    PERS robtarget YM61S:=[[-152,-102.434,331.364],[0.59149,-0.387784,-0.59121,0.3876],[-1,1,-3,0],[9E+09,8.10884,-48.3912,9E+09,9E+09,9E+09]];
    PERS robtarget YM61E:=[[-152,-136.732,324.386],[0.59149,-0.387784,-0.59121,0.3876],[-1,1,-3,0],[9E+09,8.10884,-48.3912,9E+09,9E+09,9E+09]];
    PERS robtarget YM62S:=[[-152,-143.638,394.581],[0.591293,-0.387692,-0.591403,0.387699],[-1,1,-3,0],[9E+09,7.68338,-48.3166,9E+09,9E+09,9E+09]];
    PERS robtarget YM62E:=[[-152,-165.995,387.902],[0.591293,-0.387692,-0.591403,0.387699],[-1,1,-3,0],[9E+09,7.68338,-48.3166,9E+09,9E+09,9E+09]];
    PERS robtarget YM63S:=[[-152,-136.961,363.19],[0.65293,-0.271555,-0.652826,0.271586],[-1,1,-3,0],[9E+09,9.82577,-48.6742,9E+09,9E+09,9E+09]];
    PERS robtarget YM63E:=[[-152,-158.994,355.019],[0.65293,-0.271555,-0.652826,0.271586],[-1,1,-3,0],[9E+09,9.82577,-48.6742,9E+09,9E+09,9E+09]];
    PERS robtarget YM67S:=[[-152,-100.439,322.029],[0.65293,-0.271555,-0.652826,0.271586],[-1,1,-3,0],[9E+09,8.96447,-48.5355,9E+09,9E+09,9E+09]];
    PERS robtarget YM67E:=[[-152,-134.61,314.453],[0.65293,-0.271555,-0.652826,0.271586],[-1,1,-3,0],[9E+09,8.96447,-48.5355,9E+09,9E+09,9E+09]];
    PERS robtarget YM66S:=[[-152,-225,411.8],[0.663642,-0.282382,-0.641613,0.261097],[-1,1,-3,0],[9E+09,7.65,-44.82,9E+09,9E+09,9E+09]];
    PERS robtarget YM66E:=[[-152,-189,411.8],[0.663642,-0.282382,-0.641613,0.261097],[-1,1,-3,0],[9E+09,7.65,-44.82,9E+09,9E+09,9E+09]];
    PERS robtarget YM65S:=[[-152,-225,411.8],[0.663642,-0.282382,-0.641613,0.261097],[-1,1,-3,0],[9E+09,7.65,-44.82,9E+09,9E+09,9E+09]];
    PERS robtarget YM65E:=[[-152,-189,411.8],[0.663642,-0.282382,-0.641613,0.261097],[-1,1,-3,0],[9E+09,7.65,-44.82,9E+09,9E+09,9E+09]];
    PERS robtarget YM64S:=[[-152,-225,411.8],[0.663642,-0.282382,-0.641613,0.261097],[-1,1,-3,0],[9E+09,7.65,-44.82,9E+09,9E+09,9E+09]];
    PERS robtarget YM64E:=[[-152,-189,411.8],[0.663642,-0.282382,-0.641613,0.261097],[-1,1,-3,0],[9E+09,7.65,-44.82,9E+09,9E+09,9E+09]];
    PERS robtarget YM64KS:=[[-152,-236.712,697.465],[0.65293,-0.271555,-0.652826,0.271586],[-1,1,-3,0],[9E+09,1.26795,-46.7321,9E+09,9E+09,9E+09]];
    PERS robtarget YM64KE:=[[-152,-260.629,694.325],[0.65293,-0.271555,-0.652826,0.271586],[-1,1,-3,0],[9E+09,1.26795,-46.7321,9E+09,9E+09,9E+09]];
    PERS robtarget YM65KS:=[[-152,-226.703,599.049],[0.65293,-0.271555,-0.652826,0.271586],[-1,1,-3,0],[9E+09,6,-48,9E+09,9E+09,9E+09]];
    PERS robtarget YM65KE:=[[-152,-249.965,589.663],[0.65293,-0.271555,-0.652826,0.271586],[-1,1,-3,0],[9E+09,6,-48,9E+09,9E+09,9E+09]];
    PERS robtarget YM66KS:=[[-152,-204.477,493.494],[0.65293,-0.271555,-0.652826,0.271586],[-1,1,-3,0],[9E+09,11.127,-48.873,9E+09,9E+09,9E+09]];
    PERS robtarget YM66KE:=[[-152,-226.433,477.965],[0.65293,-0.271555,-0.652826,0.271586],[-1,1,-3,0],[9E+09,11.127,-48.873,9E+09,9E+09,9E+09]];
    PERS robtarget YM67KS:=[[-152,-206.596,501.506],[0.65293,-0.271555,-0.652826,0.271586],[-1,1,-3,0],[9E+09,10.6921,-48.8079,9E+09,9E+09,9E+09]];
    PERS robtarget YM67KE:=[[-152,-228.685,486.483],[0.65293,-0.271555,-0.652826,0.271586],[-1,1,-3,0],[9E+09,10.6921,-48.8079,9E+09,9E+09,9E+09]];
    PERS robtarget YM68S:=[[-152,-131.055,340.199],[0.653753,-0.269329,-0.653858,0.269329],[-1,1,-3,0],[9E+09,11.563,-48.937,9E+09,9E+09,9E+09]];
    PERS robtarget YM68E:=[[-152,-152.782,330.846],[0.653753,-0.269329,-0.653858,0.269329],[-1,1,-3,0],[9E+09,11.563,-48.937,9E+09,9E+09,9E+09]];
    PERS robtarget YM69S:=[[-152,-97.8611,310.69],[0.65091,-0.275923,-0.651211,0.275876],[-1,1,-3,0],[9E+09,9.82577,-48.6742,9E+09,9E+09,9E+09]];
    PERS robtarget YM69E:=[[-152,-131.894,302.519],[0.65091,-0.275923,-0.651211,0.275876],[-1,1,-3,0],[9E+09,9.82577,-48.6742,9E+09,9E+09,9E+09]];

    PERS robtarget XM69S:=[[-51.74,-38.43,346.47],[0.69982,-0.714319,-0.000177661,-0.000168257],[0,-1,-1,0],[9E+09,9.82577,-48.6742,9E+09,9E+09,9E+09]];
    PERS robtarget XM69E:=[[-81.74,-44.99,332.86],[0.69982,-0.714319,-0.000177665,-0.000168594],[0,-1,-1,0],[9E+09,9.82577,-48.6742,9E+09,9E+09,9E+09]];
    PERS pose SRM69X:=[[-0.305832,0.0427742,0.000274658],[1,0,0,0]];

    PERS robtarget XM61S:=[[-51.74,-14.78,-164.74],[0.707159,-0.707055,-0.000176256,-0.000169845],[-1,1,-2,0],[9E+09,8.10884,-48.3912,9E+09,9E+09,9E+09]];
    PERS robtarget XM61E:=[[-81.74,-4.2,65],[0.707159,-0.707055,-0.000175884,-0.000170178],[-1,0,-1,0],[9E+09,8.10884,-48.3912,9E+09,9E+09,9E+09]];
    PERS pose SRM61X:=[[1.22222,0.048152,0.00824738],[1,0,0,0]];

    PERS robtarget YM69air0:=[[323.43,-909.32,657.88],[0.75163,-0.489467,-0.418492,0.142614],[-1,1,-3,0],[9E+09,0,-45,9E+09,9E+09,9E+09]];
    PERS robtarget YM69air1:=[[741.26,-226.51,717.48],[0.702088,-0.433242,-0.448105,0.344349],[-1,1,-3,0],[9E+09,0,-45,9E+09,9E+09,9E+09]];
    PERS robtarget YM69air2:=[[-25.10,218.09,408.29],[0.758077,-0.477323,-0.345026,0.280071],[0,2,-3,0],[9E+09,-7.75,-44.65,9E+09,9E+09,9E+09]];

    PERS robtarget XM49S:=[[-51,-69.7,-355.45],[0.00026471,0.974449,-0.224609,-3.1544E-05],[-1,0,0,0],[9E+09,-18.2042,-49.7958,9E+09,9E+09,9E+09]];
    PERS robtarget XM49E:=[[-81.8,-49.99,-284],[0.674318,-0.67636,0.209812,0.209312],[0,-1,0,0],[9E+09,-18.2042,-49.7958,9E+09,9E+09,9E+09]];
    PERS pose SRM49X:=[[1.06467,0.0033226,3.05176E-05],[1,0,0,0]];

    PERS robtarget YM41air0:=[[322.86,-786.84,1283.97],[0.75163,-0.489467,-0.418492,0.142614],[-1,1,-3,0],[9E+09,0,0,9E+09,9E+09,9E+09]];
    PERS robtarget YM41air1:=[[438.12,-1.09,1129.17],[0.714752,-0.443018,-0.427615,0.331677],[-1,1,-3,0],[9E+09,-7.75,-44.64,9E+09,9E+09,9E+09]];
    PERS robtarget YM41air2:=[[280.06,246.13,1162.64],[0.711624,-0.440596,-0.432799,0.334891],[-1,1,-3,0],[9E+09,-7.75,-44.65,9E+09,9E+09,9E+09]];


    PERS robtarget XM69air1:=[[406.95,-323.45,691.79],[0.681158,-0.726208,-0.091705,-0.0152943],[-1,1,-2,0],[9E+09,0,0,9E+09,9E+09,9E+09]];
    PERS robtarget XM69air2:=[[201.71,-906.55,542.23],[0.865261,-0.501321,-0.00012615,-0.00020979],[-1,-1,-1,0],[9E+09,0,-45,9E+09,9E+09,9E+09]];
    PERS robtarget XM69air3:=[[201.99,-627.42,55.34],[0.865261,-0.501321,-0.000126247,-0.000209686],[0,-1,-1,0],[9E+09,18.6523,-49.8477,9E+09,9E+09,9E+09]];
CONST robtarget XM69air13:=[[466.38,-593.12,1090.02],[0.546463,0.569613,0.0273419,-0.61333],[-1,2,-5,0],[9E+09,-7.78641E-06,6.55343E-08,9E+09,9E+09,9E+09]];
CONST robtarget XM41air13:=[[343.43,-602.92,741.89],[0.834426,0.42267,-0.338231,-0.103362],[-1,1,-4,0],[9E+09,-0.487862,-2.87448,9E+09,9E+09,9E+09]];
CONST robtarget XM41air14:=[[379.39,-439.44,917.00],[0.800618,0.381354,-0.240244,-0.394798],[-1,-2,0,0],[9E+09,-0.335924,-1.97573,9E+09,9E+09,9E+09]];
PERS robtarget pathomestnatneg45degrees:=[[1642.08,-1115.70,2682.87],[0.0875938,-0.425292,0.894504,0.106378],[-1,0,-2,0],[9E+09,-3.62032,-44.8189,9E+09,9E+09,9E+09]];
PERS robtarget A30air20:=[[382.75,-479.80,640.65],[0.391305,-0.39464,-0.584209,0.591473],[-1,0,-1,0],[9E+09,5.5,-135,9E+09,9E+09,9E+09]];
PERS robtarget B33air30:=[[-67.79,-632.04,318.04],[0.164585,0.515201,-0.472181,0.696079],[-1,1,-3,0],[9E+09,-13.5,136.5,9E+09,9E+09,9E+09]];
PERS robtarget B33air40:=[[-323.48,-348.44,373.29],[0.122788,0.72187,-0.311157,0.605812],[-1,1,-3,0],[9E+09,0,135,9E+09,9E+09,9E+09]];
PERS robtarget AIRTOANCH3:=[[-8.6,-155.14,117.47],[0.263609,-0.696089,0.660491,-0.0985977],[-1,1,-2,0],[9E+09,-40,100,9E+09,9E+09,9E+09]];
PERS robtarget H18AIRTOYL69S4:=[[204.19,-4.45,429.35],[0.341759,0.582985,-0.611047,-0.412252],[-1,1,-1,0],[9E+09,13.0111,44.6842,9E+09,9E+09,9E+09]];
PERS robtarget H18AIRTOG40_1:=[[426.16,1.81,851.86],[0.361748,-0.776477,-0.217756,0.467765],[-1,2,-2,0],[9E+09,-20,-50,9E+09,9E+09,9E+09]];

PERS robtarget XL4air23:=[[691.52,-162.97,1726.77],[0.491618,-0.102439,-0.167584,-0.848371],[-1,2,0,0],[9E+09,-10.15,44.19,9E+09,9E+09,9E+09]];
CONST robtarget AIRTOT30_10:=[[762.15,413.99,710.03],[0.077116,-0.841504,-0.161316,0.509805],[0,2,-3,0],[9E+09,-24.4581,-62.5826,9E+09,9E+09,9E+09]];
PERS robtarget F90AIRTOG40_1:=[[723.59,171.68,1587.9],[0.0227694,0.706641,-0.0229355,-0.706834],[-1,2,-2,0],[9E+09,-26,-45,9E+09,9E+09,9E+09]];

    PERS robtarget XM4air23:=[[679.92,-287.42,2151.86],[0.491619,-0.10244,-0.167584,-0.848371],[-1,1,0,0],[9E+09,0,45,9E+09,9E+09,9E+09]];

    CONST robtarget YL69air3:=[[575.73,-240.27,159.13],[0.142157,0.421918,-0.892494,-0.0723355],[-1,1,-1,0],[9E+09,12.7709,44.9833,9E+09,9E+09,9E+09]];
    CONST robtarget M49air5:=[[67.09,-478.73,-557.98],[0.703183,-0.592785,-0.0745474,0.385464],[-1,-1,0,0],[9E+09,-22,-39,9E+09,9E+09,9E+09]];
    CONST robtarget B35air_1:=[[-118.21,-790.16,748.75],[0.222108,0.671312,-0.312762,0.634183],[-1,0,-3,0],[9E+09,-14.37,135,9E+09,9E+09,9E+09]];
    CONST robtarget B35air_2:=[[-474.04,-451.28,796.03],[0.222108,0.671312,-0.312762,0.634183],[-1,0,-2,0],[9E+09,-14.37,135,9E+09,9E+09,9E+09]];
    CONST robtarget A32air_1:=[[514.14,-702.66,989.84],[0.405528,-0.370817,-0.574896,0.606248],[-1,0,-1,0],[9E+09,-1.37,-125,9E+09,9E+09,9E+09]];
    CONST robtarget A32air_2:=[[289.83,-781.28,1194.82],[0.36389,-0.403742,-0.562005,0.62348],[-1,0,-1,0],[9E+09,-1.37,-125,9E+09,9E+09,9E+09]];
    CONST robtarget B32air_1:=[[-490.20,-367.22,1109.93],[0.274121,0.675425,-0.244148,0.639571],[-1,0,-2,0],[9E+09,-5.48905,135.061,9E+09,9E+09,9E+09]];
    CONST robtarget B32air_2:=[[-137.07,-805.28,1092.89],[0.265044,0.655577,-0.224708,0.67043],[-1,0,-3,0],[9E+09,0.207107,134.293,9E+09,9E+09,9E+09]];
    CONST robtarget pjhomeSTN1zeroand180degrees:=[[1508.32,-0.13,3794.95],[0.2896,-0.00402012,0.957097,-0.0089805],[0,-1,-1,0],[9E+09,-0.0499035,180.021,9E+09,9E+09,9E+09]];
    CONST robtarget VRL52:=[[22.52,-205.94,976.00],[0.523446,-0.751557,0.24068,-0.321309],[-1,1,-2,0],[9E+09,-14.1988,49.3012,9E+09,9E+09,9E+09]];
    CONST robtarget VRM58:=[[-91.58,-127.90,952.71],[0.596926,-0.358375,-0.702933,-0.145368],[-1,0,-2,0],[9E+09,-14.1988,-49.3012,9E+09,9E+09,9E+09]];
    CONST robtarget VRG37:=[[1759.44,-115.82,2299.26],[0.0849098,0.0286926,0.995945,0.00776692],[-1,1,-2,0],[9E+09,-4.82784,-44.5104,9E+09,9E+09,9E+09]];
    CONST robtarget pzerostn194:=[[97.93,1457.09,1662.03],[0.650331,-0.0562801,-0.749121,-0.112781],[0,0,0,0],[9E+09,-0.00693957,94.0524,9E+09,9E+09,9E+09]];
    PERS robtarget pairtoL46_1:=[[191.64,-867.11,2097.29],[0.475472,-0.804215,0.076122,0.348382],[-1,-1,0,0],[9E+09,-22,-39,9E+09,9E+09,9E+09]];
    PERS robtarget XA3010:=[[682.98,-298.39,1395.43],[0.907863,-0.162432,0.0630474,0.381348],[-1,-1,-1,0],[9E+09,-10,-120,9E+09,9E+09,9E+09]];
    CONST robtarget YL69air10:=[[-200.13,-1122.9,1105.9],[0.0565202,0.961932,-0.056947,0.261247],[-1,0,-2,0],[9E+09,-10.15,44.19,9E+09,9E+09,9E+09]];
    PERS robtarget AG103danger:=[[98.44,-98.06,-251.18],[0.197528,-0.384452,-0.0264323,-0.901377],[-1,1,-3,0],[9E+09,35,102,9E+09,9E+09,9E+09]];
    PERS num limit:=-42;
    PERS robtarget R100:=[[-101.31,-14.09,-203.92],[0.000217526,0.000217373,0.707106,-0.707108],[-1,1,-3,0],[9E+09,33.5,180,9E+09,9E+09,9E+09]];

    PERS num ADJTIPSRCH:=-0.00275073;
    PERS num WTIPANGLEadj:=21.5028;
    PERS pose SRaveofG11G12:=[[0,-0.0110421,0],[1,0,0,0]];


!!!!!!these are declarations for 18H family of tips!!!!!!
    PERS pose SRTIPY18HL:=[[0,0,0],[1,0,0,0]];
    PERS pose SRTIPY18HR:=[[0,0,0],[1,0,0,0]];
	CONST robtarget SPTIPY18HLE:=[[38.00,-12.70,230.00],[0.500261,-0.499982,-0.499745,0.500012],[0,1,-2,0],[9E+09,0,-90,9E+09,9E+09,9E+09]];
	CONST robtarget SPTIPY18HRE:=[[-38.00,-12.70,230.00],[0.500261,-0.499982,0.499745,-0.500012],[0,2,-3,0],[9E+09,0,90,9E+09,9E+09,9E+09]];

	CONST robtarget SPU600HLE:=[[38,-16.5,230],[0.500261,-0.499982,-0.499745,0.500012],[0,1,-2,0],[9E+09,0,-90,9E+09,9E+09,9E+09]];
	CONST robtarget SPU650HRE:=[[-38,-16.5,230],[0.500261,-0.499982,0.499745,-0.500012],[0,2,-3,0],[9E+09,0,90,9E+09,9E+09,9E+09]];

    PERS robtarget halfwayhome_M:=[[323.43,-909.32,657.88],[0.75163,-0.489467,-0.418492,0.142614],[-1,0,-2,0],[9E+09,0,-45,9E+09,9E+09,9E+09]];
    PERS robtarget halfwayhome_L:=[[285.94,-356.45,959.29],[0.0234875,-0.737204,0.674708,-0.0273506],[-1,0,-1,0],[9E+09,0,45,9E+09,9E+09,9E+09]];
    PERS robtarget halfwayhome_A:=[[496.89,-178.24,594.79],[0.00515288,-0.986648,-0.155581,-0.0479021],[-1,2,-2,1],[9E+09,0,-135,9E+09,9E+09,9E+09]];
    PERS robtarget halfwayhome_B:=[[-434.18,-117.02,196.36],[0.0151057,0.00487122,0.994314,0.105302],[0,1,-1,0],[9E+09,0,135,9E+09,9E+09,9E+09]];
    PERS robtarget halfwayhome_G:=[[-643.51,-162.5,668.83],[0.0892073,-0.589525,0.793761,-0.120189],[-1,0,0,0],[9E+09,0,45,9E+09,9E+09,9E+09]];
    PERS robtarget halfwayhome_H:=[[780.67,-310.30,634.14],[0.236488,0.969948,0.0278582,0.0499801],[-1,1,-1,0],[9E+09,0,-45,9E+09,9E+09,9E+09]];

    PERS robtarget Troot1:=[[99.82,-61.36,159.35],[0.627626,-0.443283,-0.355925,-0.531886],[-1,0,-2,0],[9E+09,42,0,9E+09,9E+09,9E+09]];
    PERS robtarget Troot2:=[[-93.69,-61.65,160.34],[0.627627,-0.443282,-0.355926,-0.531886],[-1,0,-2,0],[9E+09,42,-7.12501E-05,9E+09,9E+09,9E+09]];

    CONST num FBfirst:=-17;
    CONST num FBsecond:= -11;

!!!!!!!!!!!!!!!!!!!!!!!!!!!!!!!!!!!END OF DECLARATIONS      !!!!!!!!!!!!!!!!!!!!!!!!!!!!!!

    CONST robtarget pat45negair1:=[[380.92,-801.85,1168.30],[0.000430871,-0.974447,0.224617,-5.83607E-05],[-1,0,0,0],[9E+09,0,-45,9E+09,9E+09,9E+09]];

    CONST robtarget AIRU1:=[[144.96,-753.41,659.47],[0.235813,-0.732282,-0.251047,0.587478],[0,2,-3,0],[9E+09,-7.00985,-63.2077,9E+09,9E+09,9E+09]];
    PERS robtarget SPUY33E:=[[-170.365,-78.7078,203.558],[0.510017,0.49007,-0.509654,-0.489864],[0,0,-3,0],[9E+09,27.0001,-45.0004,9E+09,9E+09,9E+09]];
    PERS robtarget SPUX33E:=[[-124.148,-21.7897,284.454],[0.49981,-0.500212,-0.4998,-0.500178],[-1,0,-2,0],[9E+09,27.0001,-45,9E+09,9E+09,9E+09]];
    PERS robtarget SPTY33E:=[[150.444,-80.007,203.769],[0.494322,-0.505307,0.494754,-0.505499],[0,4,-5,0],[9E+09,27,45.0002,9E+09,9E+09,9E+09]];
    PERS robtarget SPTX33E:=[[120.8,-22.1731,284.337],[0.502915,-0.503196,-0.49696,-0.496892],[-1,1,-3,0],[9E+09,26.9999,45.0001,9E+09,9E+09,9E+09]];

    PERS robtarget SPUY36E:=[[-172.488,-16.8208,232.206],[0.632719,-0.315721,-0.632589,0.315941],[0,0,-1,0],[9E+09,-15.9999,-135,9E+09,9E+09,9E+09]];
    PERS robtarget SPUX36E:=[[-142.33,-74.3,308.23],[0.6415,-0.26243,-0.650252,-0.311097],[-1,0,-2,0],[9E+09,22,-48.8794,9E+09,9E+09,9E+09]];
    PERS robtarget SPTY36E:=[[171.992,-18.0388,231.844],[0.315314,0.632751,0.315517,0.632971],[0,1,-3,0],[9E+09,-15.9999,-225,9E+09,9E+09,9E+09]];
    PERS robtarget SPTX36E:=[[142.09,-74.99,306.8],[0.313457,-0.650452,-0.267257,-0.638146],[-1,1,-2,0],[9E+09,22,48.0666,9E+09,9E+09,9E+09]];

    PERS robtarget SPUZ33E:=[[-86.4363,-72.1286,298.144],[0.606826,-0.362533,-0.518582,-0.481046],[-1,0,-2,0],[9E+09,27,-45.0002,9E+09,9E+09,9E+09]];
    PERS robtarget SPTZ33E:=[[88.1341,-70.1934,299.996],[0.431359,-0.56032,-0.305384,-0.637739],[-1,1,-3,0],[9E+09,27,44.9999,9E+09,9E+09,9E+09]];
    PERS robtarget airTIP33Z1:=[[0,-365.96,312.34],[0.549536,-0.444905,-0.444984,-0.549599],[0,-1,-1,0],[9E+09,35,0,9E+09,9E+09,9E+09]];

    PERS pose SRT33Y:=[[0.0488434,1.93963,-0.0151062],[1,0,0,0]];
    PERS pose SRT33X:=[[2.69846,0.00642776,0.032959],[1,0,0,0]];
    PERS pose SRU33Y:=[[0.00515747,-1.50801,0.0724792],[1,0,0,0]];
    PERS pose SRU33X:=[[0.709114,-0.0346451,0.0375366],[1,0,0,0]];
    PERS pose SRU33Z:=[[0.69796,-0.00751495,2.20923],[1,0,0,0]];
    PERS pose SRT33Z:=[[2.66072,0.0355301,-2.16266],[1,0,0,0]];

    PERS pose SRT36Y:=[[0.00430298,1.93455,0.0100708],[1,0,0,0]];
    PERS pose SRT36X:=[[0,0,0],[1,0,0,0]];
    PERS pose SRU36Y:=[[-0.00396729,-1.19111,-0.0218506],[1,0,0,0]];
    PERS pose SRU36X:=[[0,0,0],[1,0,0,0]];


    PERS pose SRU33XYZ:=[[0.709114,-1.50801,2.20923],[1,0,0,0]];
    PERS pose SRT33XYZ:=[[2.69846,1.93963,-2.16266],[1,0,0,0]];
    PERS pose SRU36XYZ:=[[0.709114,-1.19111,2.20923],[1,0,0,0]];
    PERS pose SRT36XYZ:=[[2.69846,1.93455,-2.16266],[1,0,0,0]];


   CONST robtarget panicpoint1:=[[381.48,-631.83,978.20],[0.486099,-0.513397,-0.48629,0.513472],[-1,-1,-1,0],[9E+09,0.918861,-133.419,9E+09,9E+09,9E+09]];
   CONST robtarget pairanchor11:=[[501.72,-592.57,-157.45],[0.699758,-0.406601,-0.58027,-0.0911068],[-1,0,-2,0],[9E+09,-5.66742,-42.0674,9E+09,9E+09,9E+09]];
   CONST robtarget pjtoparkSTA1ninety:=[[97.93,1457.09,1662.03],[0.650332,-0.0562803,-0.74912,-0.112781],[0,0,0,0],[9E+09,0.000148101,90,9E+09,9E+09,9E+09]];
   CONST robtarget pairnopinchanchor:=[[-17.24,473.18,13.73],[0.489634,0.72609,0.146511,0.459985],[-1,0,-3,0],[9E+09,6.7021,137.085,9E+09,9E+09,9E+09]];
   CONST robtarget pjhomeSTA1zeroand180degrees:=[[1508.31,-0.14,3794.91],[0.289571,-0.00401337,0.957106,-0.0089659],[-1,0,-1,0],[9E+09,0,179.985,9E+09,9E+09,9E+09]];
CONST robtarget p41air09:=[[59.75,168.19,535.47],[0.719256,-0.481993,-0.415586,0.278641],[-1,1,-3,0],[9E+09,-0.27526,-46.2246,9E+09,9E+09,9E+09]];


!!!!!!!!!!!!!!!!!!!!!!!!!!!!!!!!!!!END OF DECLARATIONS      !!!!!!!!!!!!!!!!!!!!!!!!!!!!!!

  PROC ADJWrapperROOTWIDTH18H()
        Adjustit:
         IF seamparR1.RootWidth < 0 THEN
	    seamparR1.RootWidth:= seamparR1.RootWidth*(-1);
        seamparR1.Area:= 50;
        seamparR1.Width:= 7;

        ENDIF

  ENDPROC

	PROC zRESET_Piv2Fwrap_Gse()
         !!!!!!!new...04-22-19!!!!!!!
         Piv2Fwrap_GE := Piv2Fwrap_GS;
         Piv2Fwrap_HS := Piv2Fwrap_GS;
         Piv2Fwrap_HE := Piv2Fwrap_GS;
         Piv2Fwrap_GE.trans.x := 0;
         Piv2Fwrap_HS.trans.x := Piv2Fwrap_GS.trans.x *(-1);
         Piv2Fwrap_HE.trans.x := -10;
        WaitTime\InPos, .2;
	ENDPROC

    PROC WELDFRONTWRAPpivotandtip()
        !!!!!!!!!REVISED 03-16-18 Y search first, then Z!!!!!!!!!!!
        !!!!!!!!!REVISED 03-20-18 little x move added for clearance!!!!!!!!!!!
        !!!!!!!!!REVISED 04-11-18 taught back in a Y search for the top of the pivot, switched the X disp from SR_PIV180_EDGE to SR_Piv_X!!!04-11-18!!!!!!
        ActUnit STN1;
	    AccSet 40, 40;
	    MoveJ pjthomeSTA1zero, vCellSpeed, fine, tWeldGun\WObj:=wobj0;
	    MoveJ pjhomeSTA1zeroand180degrees, vCellSpeed, fine, tWeldGun\WObj:=wobj0;
	    TPErase;
        PDispOff;
        Piv_YZ180_Xset;
        MoveJ Offs(SP_PIV180_XS,-100,600,0), V500, z5, tWeldGun\WObj:=wobjHsideplate;
        MoveL offs(SP_PIV180_XS,-50,50,0), V500, z5, tWeldGun\WObj:=wobjHsideplate;
        Search_1D SR_Piv_X\SearchStop:=PivFOUND_X, SP_PIV180_XS, SP_PIV180_XE, v300, tWeldGun\WObj:=wobjHsideplate\SchSpeed:=10;
        Piv_YZ180_Xset;
        TPWrite "SR_Piv_X XYZ:="\Pos:=SR_Piv_X.trans;
        MoveL offs(SP_PIV180_XE,-50,0,0), V500, z5, tWeldGun\WObj:=wobjHsideplate;
        MoveL offs(SP_PIV180_XE,-50,0,100), V500, z5, tWeldGun\WObj:=wobjHsideplate;
        MoveL Offs(SP_Piv180_Xe,-150,0,100), V500, z5, tWeldGun\WObj:=wobjHsideplate;
        YfirstthenZ:
        MoveJ offs(SP_Piv180_Ys,0,300,0), V500, z5, tWeldGun\WObj:=wobjHsideplate;
        MoveL offs(SP_Piv180_Ys,0,50,0), V500, z5, tWeldGun\WObj:=wobjHsideplate;
        Search_1D SR_Piv_Y\SearchStop:=PivFOUND_Y, SP_Piv180_Ys, SP_Piv180_Ye, v300, tWeldGun\WObj:=wobjHsideplate\SchSpeed:=10;
        TPWrite "SR_Piv_Y0 XYZ:="\Pos:=SR_Piv_Y.trans;
        MoveL PivFOUND_Y, V500, z1, tWeldGun\WObj:=wobjHsideplate;
        PDispOff;
        WaitTime\InPos, 1;
        PivFOUND_Y := CRobT(\Tool:=tWeldGun\WObj:=obSTN1);
        WaitTime\InPos, 1;
        MoveJ offs(SP_Piv180_Ys,0,350,0), V500, z1, tWeldGun\WObj:=wobjHsideplate;
        nowz:
        MoveJ Offs(SP_Piv180_Zs,0,300,20), V500, z1, tWeldGun\WObj:=wobjHsideplate;
        MoveL offs(SP_Piv180_Zs,0,0,20), V500, z1, tWeldGun\WObj:=wobjHsideplate;
        Search_1D SR_Piv_Z\SearchStop:=PivFOUND_Z, SP_Piv180_Zs, SP_Piv180_Ze, v300, tWeldGun\WObj:=wobjHsideplate\PrePDisp:=SR_Piv_Y\SchSpeed:=10;
        TPWrite "SR_Piv_Z XYZ:="\Pos:=SR_Piv_Z.trans;
        MoveL PivFOUND_Z, V500, z1, tWeldGun\WObj:=wobjHsideplate;
        PDispOff;
        WaitTime\InPos, 1;
        PivFOUND_Z := CRobT(\Tool:=tWeldGun\WObj:=obSTN1);
        WaitTime\InPos, 1;
        MoveL offs(SP_Piv180_Zs,0,0,50), V500, z10, tWeldGun\WObj:=wobjHsideplate;
        MoveL offs(SP_Piv180_Zs,0,300,100), V500, z20, tWeldGun\WObj:=wobjHsideplate;
        PivWobj_Translation_Locator wobj_PivCam, PivFOUND_Y, PivFOUND_Z, WPIVOTANGLE;
        WaitTime\InPos, 1;
        PivWobj_Rotation_Locator PivFOUND_Y, PivFOUND_Z, wobj_PivCam;
	    WaitTime\InPos, 1;
        MoveJ offs(Piv2Fwrap_RS,0,350,0), V500, z1, tWeldGun\WObj:=wobj_PivCam;
        !!!!!!!! new Y SEARCH  HERE 4-11-18!!!!!!
		MoveJ Offs(SPR5E,0,200,0), v500, z5, tWeldGun\WObj:=wobj_PivCam;
		MoveL Offs(SPR5E,0,50,0), v500, z1, tWeldGun\WObj:=wobj_PivCam;
        Search_1D SRR1Y, Offs(SPR5E,0,30,0), SPR5E, v200, tWeldGun\WObj:=wobj_PivCam\SchSpeed:=10;
		MoveL Offs(SPR5E,0,50,0), v200, z5, tWeldGun\WObj:=wobj_PivCam;
		MoveJ Offs(SPR5E,0,200,0), v500, z5, tWeldGun\WObj:=wobj_PivCam;
        !!!!!!!!PUT THE new Y SEARCH  HERE 4-11-18!!!!!!
        MoveJ Offs(SP_PIV180_JOINT_S,0,200,0), vExtMax, z5, tWeldGun\WObj:=wobj_PivCam;
	    MoveL Offs(SP_PIV180_JOINT_S,0,100,0), vExtMax, z5, tWeldGun\WObj:=wobj_PivCam;
	    PDispOff;
        TPErase;
        Search_Edge\TopCornerDisp:=SR_PIV180_EDGE, Offs(SP_PIV180_EDGE_E,0,0,-15), SP_PIV180_EDGE_E, edgedataR10\InitSchL:=15\Spacing:=2\PackStart, v50, tWeldGun\WObj:=wobj_PivCam\PrePDisp:=SRRY1\SrchSpeed:=5;
        TPWrite "SR_PIV180_EDGE XYZ:="\Pos:=SR_PIV180_EDGE.trans;
	    MoveL Offs(SP_PIV180_JOINT_S,0,100,0), v200, z5, tWeldGun\WObj:=wobj_PivCam;
        TPErase;
        Search_Joint SR_PIV180_JOINT, Offs(SP_PIV180_JOINT_E,0,0,-15), SP_PIV180_JOINT_E, bevelparamR1, seamparR1\InitSchL:=15\PackStart, v50, tWeldGun\WObj:=wobj_PivCam\SrchSpeed:=5;
        TPWrite "SR_PIV180_JOINT XYZ:="\Pos:=SR_PIV180_JOINT.trans;
	    PDispOff;
		!Stop;
        ADJWrapperROOTWIDTH18H;
		MoveL Offs(SP_PIV180_JOINT_E,0,100,0), vExtMax, z5, tWeldGun\WObj:=wobj_PivCam;
		MoveL Offs(SP_PIV180_JOINT_E,0,200,0), vExtMax, z5, tWeldGun\WObj:=wobj_PivCam;
		MoveJ Offs(SP_PIV180_JOINT_E,0,800,0), vExtMax, z5, tWeldGun\WObj:=wobj_PivCam;
        !!!!!  GOING TO THE TIP   !!!!!!!
        MoveJ Offs(SPP1E,0,400,50), v500, z5, tWeldGun\WObj:=wobjHtip;
		MoveJ Offs(SPP2E,0,200,0), vExtMax, z5, tWeldGun\WObj:=wobjHtip;
		PDispOff;
        TPErase;
        Search_1D SRPY, Offs(SPP2E,0,20,0), SPP2E, v200, tWeldGun\WObj:=wobjHtip\SchSpeed:=10;
        TPWrite "SRPY XYZ:="\Pos:=SRPY.trans;
		MoveL Offs(SPP2E,0,20,0), v200, z5, tWeldGun\WObj:=wobjHtip;
		MoveJ Offs(SPP2E,0,200,0), vExtMax, z5, tWeldGun\WObj:=wobjHtip;
		MoveJ Offs(SPP1E,0,400,50), vExtMax, z5, tWeldGun\WObj:=wobjHtip;
		MoveJ Offs(SPP1E,0,200,50), vExtMax, z5, tWeldGun\WObj:=wobjHtip;
		MoveL Offs(SPP1E,0,50,20), vExtMax, z5, tWeldGun\WObj:=wobjHtip;
		MoveL RelTool(SPP1E,0,-15,-50), v100, z1, tWeldGun\WObj:=wobjHtip;
        TPErase;
        Search_Edge\TopCornerDisp:=SRP1, Offs(SPP1E,0,0,15), SPP1E, edgedataPQ1\InitSchL:=15\Spacing:=2\PackStart, v50, tWeldGun\WObj:=wobjHtip\SrchSpeed:=5;
        TPWrite "SRP1 XYZ:="\Pos:=SRP1.trans;
		MoveL RelTool(SPP1E,0,-15,-50), v100, z1, tWeldGun\WObj:=wobjHtip;
		MoveL Offs(SPP1E,0,50,20), vExtMax, z5, tWeldGun\WObj:=wobjHtip;
		MoveL Offs(SPP3E,30,200,0), vExtMax, z5, tWeldGun\WObj:=wobjHtip;
        TPErase;
        Search_1D SRPX, Offs(SPP3E,30,0,0), SPP3E, v200, tWeldGun\WObj:=wobjHtip\SchSpeed:=10;
        TPWrite "SRPX XYZ:="\Pos:=SRPX.trans;
		MoveL Offs(SPP3E,30,0,0), v200, z5, tWeldGun\WObj:=wobjHtip;
		MoveL Offs(SPP3E,30,200,0), vExtMax, z5, tWeldGun\WObj:=wobjHtip;
		MoveL Offs(SPP3E,30,250,0), vExtMax, z5, tWeldGun\WObj:=wobjHtip;
		MoveJ Offs(SPP3E,90,750,0), vExtMax, z5, tWeldGun\WObj:=wobjHtip;
		PDispOff;
		MoveJ Offs(Piv2Fwrap_RS,-80,550,0), vExtMax, z5, tWeldGun\WObj:=wobj_PivCam;
		MoveJ Offs(Piv2Fwrap_RS,-80,200,0), vExtMax, z5, tWeldGun\WObj:=wobj_PivCam;
        TPErase;
!!!!!!!!!!!!!THESE assigns are changed 04-11-18!!!!!!!!
        SR_PIV180_JOINT.trans.X := SR_Piv_X.trans.X;
		SR_PIV180_EDGE.trans.X := SR_Piv_X.trans.X;
        SR_PIV180_EDGE.trans.Y := SRRY1.trans.Y;
        SR_PIV180_JOINT.trans.Y := SRRY1.trans.Y;
!!!!!!!!!!!!!!!!!!!!!!!!!!!!!!!!!!!!!!!!!!!
!!!!!!!!!!!!!!!!!!!new 02-27-29!!!!!!!!!!!!!!!!!!!!!!
        Piv2Fwrap_RS.extax.eax_b:= Piv2Fwrap_GS.extax.eax_b - 9;
        Piv2Fwrap_RE.extax.eax_b := Piv2Fwrap_GS.extax.eax_b - 9;
	    WaitTime\InPos, 0.3;
!!!!!!!!!!!!!!!!!!!!!!!!!!!!!!!!!!!!!!!!!!!
		!Stop;
        !zRESET_Piv2Fwrap_Gse;
		!Stop;
        PDispSet SR_PIV180_EDGE;
		ArcLStart Piv2Fwrap_RS, v100, smPQRSroot, wdR1R2root\Weave:=wv0, z1, tWeldGun\WObj:=wobj_PivCam;
		ArcLEnd Piv2Fwrap_RE, v100, smPQRSroot, wdR1R2root\Weave:=wv0, z1, tWeldGun\WObj:=wobj_PivCam;
		PDispOff;
		MoveL offs(Piv2Fwrap_RE,0,100,0), v500, z5, tWeldGun\WObj:=wobj_PivCam;
        TPErase;
        TPWrite "NOW WORKING ON WELD 'R' (2nd pass)";
		MoveL Offs(Piv2FWrap_GS,0,100,0), v200, z5, tWeldGun\WObj:=wobj_PivCam;
		seamparS1 := seamparR1;
		seamparS1.SeamName := "SWELD";
        PDispSet SR_PIV180_JOINT;
        HWeldStart Piv2Fwrap_GS, seamparR1, smRS1, wdR5R6cover\Weave:=wvR5R6cover, v100, z1, tWeldGun\WObj:=wobj_PivCam\Track:=trRS56;
		HWeldLEnd Piv2Fwrap_GE, seamparR1, v100, z1, tWeldGun\WObj:=wobj_PivCam;
		MoveL RelTooL(Piv2Fwrap_GE,0,0,-50), vExtMax, z1, tWeldGun\WObj:=wobj_PivCam;
		HWeldStart Piv2Fwrap_HS, seamparS1, smRS1, wdR5R6cover\Weave:=wvR5R6cover, v100, z1, tWeldGun\WObj:=wobj_PivCam\Track:=trRS56;
		HWeldLEnd Piv2Fwrap_HE, seamparS1, v100, z1, tWeldGun\WObj:=wobj_PivCam;
        MoveJ Offs(Piv2Fwrap_HE,0,200,0), vExtMax, z5, tWeldGun\WObj:=wobj_PivCam;
        TPErase;
        TPWrite "NOW WORKING ON WELD 'R' (final pass)";
		GOTO TAKE;
        HWReplay\Start\End, layRWELD, smRS1, wdR5R6cover, wvR5R6cover, v200, z1, tWeldGun\WObj:=wobj_PivCam;
		HWReplay\Start\End, laySWELD, smRS1, wdR5R6cover, wvR5R6cover, vExtMax, z1, tWeldGun\WObj:=wobj_PivCam;
        TAKE:
		PDispOff;
        TPErase;
        TPWrite "NOW WORKING ON WELD 'P'";
		MoveL Offs(Piv2Fwrap_HE,0,200,0), vExtMax, z5, tWeldGun\WObj:=wobj_PivCam;
		MoveL Offs(Piv2Fwrap_HE,0,600,0), vExtMax, z5, tWeldGun\WObj:=wobj_PivCam;
		MoveJ Offs(P1,0,300,200), vExtMax, z5, tWeldGun\WObj:=wobjHtip;
		MoveL RelTool(P2,0,-20,-20), v100, z1, tWeldGun\WObj:=wobjHtip;
		MoveL RelTool(P2,0,0,-20), v100, z1, tWeldGun\WObj:=wobjHtip;
		PDispOff;
		SRP1.trans.y := SRPY.trans.y;
		SRP1.trans.x := SRPX.trans.x;
        !Stop;
        !!!!CHECK THESE (2) WELDS
        !!!!DELETE THIS STOP
		rootadded:
		PDispSet SRP1;
		ArcLStart Offs(P2,6,0,0), v100, smpqroot, wdP1Q1root\Weave:=wv0, z1, tWeldGun\WObj:=wobjHtip;
		ArcLEnd Offs(P1,-6,0,0), v100, smpqroot, wdP1Q1root\Weave:=wv0, z1, tWeldGun\WObj:=wobjHtip;
		MoveL Offs(P2E,0,50,20), vExtMax, z5, tWeldGun\WObj:=wobjHtip;
		ArcLStart Offs(Q2,-6,0,0), v100, smpqroot, wdP1Q1root\Weave:=wv0, z1, tWeldGun\WObj:=wobjHtip;
		ArcLEnd Offs(Q1,6,0,0), v100, smpqroot, wdP1Q1root\Weave:=wv0, z1, tWeldGun\WObj:=wobjHtip;
		MoveL Offs(P2E,0,50,20), vExtMax, z5, tWeldGun\WObj:=wobjHtip;
		WaitTime\InPos, 6;
		PDispSet SRP1;
		ArcLStart P2, v100, smPQ1, wdP1Q1cover\Weave:=wvP1Q1cover, z1, tWeldGun\WObj:=wobjHtip;
		ArcLEnd P2E, v100, smPQ1, wdP1Q1cover\Weave:=wvP1Q1cover, z1, tWeldGun\WObj:=wobjHtip;
		MoveL Offs(P2E,0,50,20), vExtMax, z5, tWeldGun\WObj:=wobjHtip;
		ArcLStart P1, v100, smPQ1, wdP1Q1cover\Weave:=wvP1Q1cover, z1, tWeldGun\WObj:=wobjHtip;
		ArcLEnd P1E, v100, smPQ1, wdP1Q1cover\Weave:=wvP1Q1cover, z1, tWeldGun\WObj:=wobjHtip;
		MoveL Offs(P1E,0,100,20), vExtMax, z5, tWeldGun\WObj:=wobjHtip;
        TPErase;
        TPWrite "NOW WORKING ON WELD 'Q'";
		MoveJ Offs(Q2,0,50,20), vExtMax, z5, tWeldGun\WObj:=wobjHtip;
		PDispSet SRP1;
		ArcLStart Q2, v100, smPQ1, wdP1Q1cover\Weave:=wvP1Q1cover, z1, tWeldGun\WObj:=wobjHtip;
		ArcLEnd Q2E, v100, smPQ1, wdP1Q1cover\Weave:=wvP1Q1cover, z1, tWeldGun\WObj:=wobjHtip;
		MoveL Offs(Q2E,0,100,20), vExtMax, z5, tWeldGun\WObj:=wobjHtip;
		ArcLStart Q1, v100, smPQ1, wdP1Q1cover\Weave:=wvP1Q1cover, z1, tWeldGun\WObj:=wobjHtip;
		ArcLEnd Q1E, v100, smPQ1, wdP1Q1cover\Weave:=wvP1Q1cover, z1, tWeldGun\WObj:=wobjHtip;
		MoveL Offs(Q1E,0,100,20), vExtMax, z5, tWeldGun\WObj:=wobjHtip;
        TPErase;
		PDispOff;
		MoveL Offs(Q2E,0,200,200), vExtMax, z5, tWeldGun\WObj:=wobjHtip;
		MoveJ pjhomeSTA1zeroand180degrees, vCellSpeed, fine, tWeldGun\WObj:=wobj0;
		MoveJ pjthomeSTA1zero, vCellSpeed, fine, tWeldGun\WObj:=wobj0;
		DONE:
    ENDPROC

 	PROC zRESET_T1112()
         !!!!!!!new...02-27-19!!!!!!!
         T12 := T11;
         U11 := T11;
         U12 := T11;
         T12.trans.x := 0;
         U11.trans.x := T11.trans.x *(-1);
         U12.trans.x := 10;
        WaitTime\InPos, .2;
	ENDPROC

	PROC WELDBACKWRAPtotip()
	    ActUnit STN1;
	    AccSet 75, 75;
	    MoveJ pjthomeSTA1zero, vCellSpeed, fine, tWeldGun\WObj:=wobj0;
	    PDispOff;
		MoveJ Offs(T12,0,-200,0), vExtMax, z5, tWeldGun\WObj:=wobjHtip;
		MoveL Offs(U11,-100,-200,0), vExtMax, z5, tWeldGun\WObj:=wobjHtip;
        TPErase;
		Search_1D\Wire, SRT12X, SPT12S, SPT12E, v200, tWeldGun\WObj:=wobjHtip\SchSpeed:=10;
        TPWrite "SRT12X XYZ:="\Pos:=SRT12X.trans;
		MoveL Offs(U11,-100,-200,0), vExtMax, z5, tWeldGun\WObj:=wobjHtip;
		MoveL Offs(T12,0,-200,0), vExtMax, z5, tWeldGun\WObj:=wobjHtip;
	    MoveL Offs(T12,0,-40,0), vExtMax, z5, tWeldGun\WObj:=wobjHtip;
	    PDispOff;
	    Search_Edge\TopCornerDisp:=T55, SPT55S, SPT55E, edgedataT55\InitSchL:=15\Spacing:=2\PackStart, v50, tWeldGun\WObj:=wobjHtip\SrchSpeed:=5;
        TPWrite "T55 XYZ:="\Pos:=T55.trans;
	    MoveL Offs(T11,-30,-100,0), vExtMax, z5, tWeldGun\WObj:=wobjHtip;
        TPErase;
	    T55.trans.x := SRT12X.trans.x;
        TPErase;
         !Stop;
         !zRESET_T1112;
         !Stop;
        PDispSet T55;
        ArcLStart T1, v500, smTUroot, wdT1112root, fine, tWeldGun\WObj:=wobjHtip;
        ArcLEnd U1, v500, smTUroot, wdT1112root, fine, tWeldGun\WObj:=wobjHtip;
        MoveL Offs(T11,0,-200,0), vExtMax, z5, tWeldGun\WObj:=wobjHtip;
        TPWrite "NOW WORKING ON WELD 'T'";
		PDispSet T55;
		ArcLStart T11, v500, smTU, wdT1112cover\Weave:=wvT1112cover, fine, tWeldGun\WObj:=wobjHtip\Track:=trTIPBACKhiteonly;
		ArcLEnd T12, v500, smTU, wdT1112cover\Weave:=wvT1112cover, fine, tWeldGun\WObj:=wobjHtip\Track:=trTIPBACKhiteonly;
		MoveL Offs(T12,0,-100,0), vExtMax, z5, tWeldGun\WObj:=wobjHtip;
		ArcLStart U11, v500, smTU, wdT1112cover\Weave:=wvT1112cover, fine, tWeldGun\WObj:=wobjHtip\Track:=trTIPBACKhiteonly;
		ArcLEnd U12, v500, smTU, wdT1112cover\Weave:=wvT1112cover, fine, tWeldGun\WObj:=wobjHtip\Track:=trTIPBACKhiteonly;
		MoveL Offs(U12,0,-200,0), vExtMax, z5, tWeldGun\WObj:=wobjHtip;
        TPErase;
		PDispOff;
		MoveJ pjthomeSTA1zero, vCellSpeed, fine, tWeldGun\WObj:=wobj0;
		bedone:
	ENDPROC

   	PROC Piv_YZ180_Xset ()
        VAR NUM PIV_WIDTH;

        !!!!!!!!!!!!!!!!!!!!!!!!!!!!!!!!!!!!!!!!!!!!!!!!!!!!!!!!!!!!!!!!!!!!!!!!!!!!!!
        IF PIVOT_USED = 674961 OR PIVOT_USED = 350404  THEN !77F THRU 120F
              PIV_WIDTH:=  (382/2);
        ELSEIF PIVOT_USED = 6099018 THEN  !18H THRU 20H
                 PIV_WIDTH:=  (231.6/2);
        ELSEIF PIVOT_USED = 6089330 THEN  !33H
                 PIV_WIDTH:=  (292/2);
        ELSEIF PIVOT_USED = 6802774 THEN  !24H
                 PIV_WIDTH:=  (250/2);
        ELSEIF PIVOT_USED = 6870131 THEN  !38H
                 PIV_WIDTH:=  (325/2);
        ELSEIF PIVOT_USED = 6845931 THEN  !42H
                 PIV_WIDTH := (331/2);
        ENDIF

    SP_PIV180_XE.trans.X := ((PIV_WIDTH) + NOZZLE_RADIUS) * (-1) ;
    SP_PIV180_XS.trans.X := ((PIV_WIDTH) + NOZZLE_RADIUS + 50) * (-1) ;

    SP_Piv180_Ye.trans.X := PivFOUND_X.TRANS.X + NOZZLE_RADIUS * 2 ;
    SP_Piv180_Ys.trans.X := PivFOUND_X.TRANS.X + NOZZLE_RADIUS * 2 ;

    SP_Piv180_Ze.trans.X := PivFOUND_X.TRANS.X + NOZZLE_RADIUS * 2 ;
    SP_Piv180_Zs.trans.X := PivFOUND_X.TRANS.X + NOZZLE_RADIUS * 2 ;

	ENDPROC

	PROC WELDtip()
        !!BEST WELDTIP (18H) as of 04-08-18 (has XYZ searches, z shifted by x,y)!!!!!!
		ActUnit STN1;
		AccSet 40, 40;
		MoveJ pjthomeSTA1zero, vCellSpeed, fine, tWeldGun\WObj:=wobj0;
		MoveJ Offs(T50,-500,-50,100), vExtMax, z1, tWeldGun\WObj:=wobjHtip;
		PDispOff;
		TPErase;
		MoveL Offs(T50,-50,0,0), v200, z1, tWeldGun\WObj:=wobjHtip;
        TPErase;
		Search_Edge\TopCornerDisp:=SRT50, SPT50S, SPT50E, edgedataT50\InitSchL:=15\Spacing:=4\PackStart, v100, tWeldGun\WObj:=wobjHtip\SrchSpeed:=5;
        TPWrite "SRT50 XYZ:="\Pos:=SRT50.trans;
		MoveJ Offs(T50,-500,-50,100), vExtMax, z1, tWeldGun\WObj:=wobjHtip;
		MoveJ Offs(T41,500,-50,100), vExtMax, z1, tWeldGun\WObj:=wobjHtip;
		MoveL Offs(T41,50,-0,0), v200, z1, tWeldGun\WObj:=wobjHtip;
        TPErase;
		Search_Edge\TopCornerDisp:=SRT40, SPT40S, SPT40E, edgedataT40\InitSchL:=15\Spacing:=4\PackStart, v100, tWeldGun\WObj:=wobjHtip\SrchSpeed:=5;
        TPWrite "SRT40 XYZ:="\Pos:=SRT40.trans;
		MoveL Offs(T41,50,-0,0), v200, z1, tWeldGun\WObj:=wobjHtip;
		T40:
        TPErase;
        TPWrite "NOW WORKING ON WELD 'T40'";
		PDispSet SRT40;
		ArcLStart T41, v100, smT50, wdT50root\Weave:=wv0, fine, tWeldGun\WObj:=wobjHtip;
		ArcLEnd T42, v100, smT50, wdT50root\Weave:=wv0, fine, tWeldGun\WObj:=wobjHtip;
		MoveL Offs(T41,50,0,0), v200, z1, tWeldGun\WObj:=wobjHtip;
		WaitTime 8;
		ArcLStart T43, v100, smT50, wdT50\Weave:=wvT50, fine, tWeldGun\WObj:=wobjHtip;
		ArcLEnd T44, v100, smT50, wdT50\Weave:=wvT50, fine, tWeldGun\WObj:=wobjHtip;
		MoveL Offs(T41,50,-0,0), v200, z1, tWeldGun\WObj:=wobjHtip;
		PDispOff;
		MoveJ Offs(T41,500,-50,100), vExtMax, z1, tWeldGun\WObj:=wobjHtip;
        TPErase;
        TPWrite "NOW WORKING ON WELD 'T50'";
		MoveJ Offs(T50,-500,-50,100), vExtMax, z1, tWeldGun\WObj:=wobjHtip;
		MoveL Offs(T50,-50,0,0), v200, z1, tWeldGun\WObj:=wobjHtip;
		PDispSet SRT50;
		ArcLStart T50, v100, smT50, wdT50root\Weave:=wv0, fine, tWeldGun\WObj:=wobjHtip;
		ArcLEnd T51, v100, smT50, wdT50root\Weave:=wv0, fine, tWeldGun\WObj:=wobjHtip;
		MoveL Offs(T50,-50,0,0), v200, z1, tWeldGun\WObj:=wobjHtip;
		WaitTime 8;
		ArcLStart T52, v100, smT50, wdT50\Weave:=wvT50, fine, tWeldGun\WObj:=wobjHtip;
		ArcLEnd T53, v100, smT50, wdT50\Weave:=wvT50, fine, tWeldGun\WObj:=wobjHtip;
		PDispOff;
		MoveL Offs(T50,-50,0,0), v200, z1, tWeldGun\WObj:=wobjHtip;
		MoveJ Offs(T50,-500,-50,100), vExtMax, z1, tWeldGun\WObj:=wobjHtip;
		IF bANC2CLOSE2_TIP = TRUE THEN
			TPWrite "ANCHOR IS TOO CLOSE TO TIP, WELD THAT BY HAND'";
			MoveJ AIRTOT30_3, vExtMax, z1, tWeldGun\WObj:=wobjHtip;
			GOTO SKIP_TU30s;
		ELSE
			GOTO KEEPGOING;
		ENDIF
        KEEPGOING:
        TPErase;
        TPWrite "NOW WORKING ON WELD 'T30'";
		MoveJ Offs(T50,-500,-50,100), vExtMax, z1, tWeldGun\WObj:=wobjHtip;
		MoveJ pjthomeSTA1zero, vCellSpeed, fine, tWeldGun\WObj:=wobj0;
		CutWire;
		ActUnit STN1;
		AccSet 40, 40;
		MoveJ pjthomeSTA1zero, vCellSpeed, fine, tWeldGun\WObj:=wobj0;
		SEARCHTIPears:
		MoveJ Offs(U33,150,-300,0), vExtMax, z1, tWeldGun\WObj:=wobjHtip;
        SEARCHU33Y:
		MoveJ Offs(SPUY33E,0,-100,0), vExtMax, z1, tWeldGun\WObj:=wobjHtip;
		Search_1D SRU33Y, RelTool(SPUY33E,20,0,0), SPUY33E, v50, tWeldGun\WObj:=wobjHtip\SchSpeed:=10;
		MoveJ Offs(SPUY33E,0,-100,0), v200, z1, tWeldGun\WObj:=wobjHtip;
		MoveJ Offs(U33,150,-300,0), vExtMax, z1, tWeldGun\WObj:=wobjHtip;
		MoveL Offs(U33,-250,-300,0), vExtMax, z1, tWeldGun\WObj:=wobjHtip;
        SEARCHU33X:
		MoveL Offs(SPUX33E,-80,0,0), vExtMax, z1, tWeldGun\WObj:=wobjHtip;
		Search_1D SRU33X, Offs(SPUX33E,-30,0,0), SPUX33E, v50, tWeldGun\WObj:=wobjHtip\SchSpeed:=10;
		MoveL Offs(SPUX33E,-80,0,0), v200, z1, tWeldGun\WObj:=wobjHtip;
		MoveL Offs(U33,-250,-300,0), vExtMax, z1, tWeldGun\WObj:=wobjHtip;
		MoveJ Offs(U33,150,-300,0), vExtMax, z1, tWeldGun\WObj:=wobjHtip;
		!MoveL Offs(U33,50,-50,0), v200, z1, tWeldGun\WObj:=wobjHtip;
		SRU33XYZ.trans.x := SRU33X.trans.x;
		SRU33XYZ.trans.y := SRU33Y.trans.y;
		!MoveJ airTIP33Z1, vExtMax, fine, tWeldGun\WObj:=wobjHtip;
		searchUZ:
		MoveL Offs(SPUZ33E,30,-30,30), v200, z1, tWeldGun\WObj:=wobjHtip;
		Search_1D SRU33Z, Offs(SPUZ33E,0,0,20), SPUZ33E, v50, tWeldGun\WObj:=wobjHtip\PrePDisp:=SRU33X\SchSpeed:=10;
		TPWrite "SRU33Z XYZ:="\Pos:=SRU33Z.trans;
		MoveL Offs(SPUZ33E,30,-30,30), v200, z1, tWeldGun\WObj:=wobjHtip;
		SRU33XYZ.trans.z := SRU33Z.trans.z;
        WaitTime\InPos, .1;
		PDispSet SRU33XYZ;
		ArcLStart U33, v100, smTU3031quick2, wdTU3031quick2\Weave:=wvTU3031quick2, fine, tWeldGun\WObj:=wobjHtip\Track:=trTIPears;
		ArcL U34, v100, smTU3031quick2, wdTU3031quick2\Weave:=wvTU3031quick2, z10, tWeldGun\WObj:=wobjHtip\Track:=trTIPears;
		ArcLEnd U35, v100, smTU3031quick2, wdTU3031quick2\Weave:=wvTU3031quick2, z10, tWeldGun\WObj:=wobjHtip\Track:=trTIPears;
		PDispOff;
		MoveL Offs(U33,50,-50,0), v200, z1, tWeldGun\WObj:=wobjHtip;
		MoveL Offs(U33,150,-300,0), vExtMax, z1, tWeldGun\WObj:=wobjHtip;
		MoveJ pjthomeSTA1zero, vCellSpeed, fine, tWeldGun\WObj:=wobj0;
		CutWire;
		ActUnit STN1;
		AccSet 40, 40;
		MoveJ pjthomeSTA1zero, vCellSpeed, fine, tWeldGun\WObj:=wobj0;
		!MoveL Offs(T33,-150,-300,0), vExtMax, z1, tWeldGun\WObj:=wobjHtip;
		MoveJ Offs(T33,0,-500,0), vExtMax, z1, tWeldGun\WObj:=wobjHtip;
        SEARCHT33Y:
		MoveJ Offs(SPTY33E,0,-200,0), vExtMax, z1, tWeldGun\WObj:=wobjHtip;
		Search_1D SRT33Y, RelTool(SPTY33E,20,0,0), SPTY33E, v50, tWeldGun\WObj:=wobjHtip\SchSpeed:=10;
		MoveL Offs(SPTY33E,0,-200,0), vExtMax, z1, tWeldGun\WObj:=wobjHtip;
		MoveJ Offs(T33,0,-500,0), vExtMax, z1, tWeldGun\WObj:=wobjHtip;
        SEARCHT33X:
		MoveL Offs(SPTX33E,80,0,0), vExtMax, z1, tWeldGun\WObj:=wobjHtip;
		Search_1D SRT33X, Offs(SPTX33E,30,0,0), SPTX33E, v50, tWeldGun\WObj:=wobjHtip\SchSpeed:=10;
		MoveL RelTool(SPTX33E,0,80,0), v200, z1, tWeldGun\WObj:=wobjHtip;
		MoveL Offs(T33,0,-500,0), vExtMax, z1, tWeldGun\WObj:=wobjHtip;
		MoveL Offs(T33,-150,-300,0), vExtMax, z1, tWeldGun\WObj:=wobjHtip;
		!MoveL Offs(T33,-50,-50,0), vExtMax, z1, tWeldGun\WObj:=wobjHtip;
		SRT33XYZ.trans.x := SRT33X.trans.x;
		SRT33XYZ.trans.y := SRT33Y.trans.y;
		searchTZ:
		MoveL Offs(SPTZ33E,-30,-30,30), v200, z1, tWeldGun\WObj:=wobjHtip;
		Search_1D SRT33Z, Offs(SPTZ33E,0,0,20), SPTZ33E, v50, tWeldGun\WObj:=wobjHtip\PrePDisp:=SRT33X\SchSpeed:=10;
		TPWrite "SRT33Z XYZ:="\Pos:=SRT33Z.trans;
		MoveL Offs(SPTZ33E,-30,-30,30), v200, z1, tWeldGun\WObj:=wobjHtip;
		!MoveJ airTIP33Z1, vExtMax, z5, tWeldGun\WObj:=wobjHtip;
		SRT33XYZ.trans.z := SRT33Z.trans.z;
        WaitTime\InPos, .1;
		PDispSet SRT33XYZ;
		ArcLStart T33, v100, smTU3031quick2, wdTU3031quick2\Weave:=wvTU3031quick2, fine, tWeldGun\WObj:=wobjHtip\Track:=trTIPears;
		ArcL T34, v100, smTU3031quick2, wdTU3031quick2\Weave:=wvTU3031quick2, z10, tWeldGun\WObj:=wobjHtip\Track:=trTIPears;
		ArcLEnd T35, v100, smTU3031quick2, wdTU3031quick2\Weave:=wvTU3031quick2, z10, tWeldGun\WObj:=wobjHtip\Track:=trTIPears;
		PDispOff;
		MoveL RelTool(T33,0,0,-30), v200, z1, tWeldGun\WObj:=wobjHtip;
		MoveL RelTool(T33,0,0,-300), vExtMax, z1, tWeldGun\WObj:=wobjHtip;
		MoveJ AIRTOU30_1, vExtMax, z1, tWeldGun\WObj:=wobjHtip;
		MoveL RelTool(U36,0,0,-300), vExtMax, z1, tWeldGun\WObj:=wobjHtip;
        SEARCHU36Y:
		MoveL Offs(SPUY36E,0,100,0), vExtMax, z1, tWeldGun\WObj:=wobjHtip;
		Search_1D SRU36Y, Offs(SPUY36E,0,20,0), SPUY36E, v100, tWeldGun\WObj:=wobjHtip\SchSpeed:=10;
		MoveL Offs(SPUY36E,0,150,0), vExtMax, z1, tWeldGun\WObj:=wobjHtip;
		SRU36XYZ.trans.x := SRU33X.trans.x;
		SRU36XYZ.trans.y := SRU36Y.trans.y;
		SRU36XYZ.trans.z := SRU33Z.trans.z;
        WaitTime\InPos, .1;
		MoveL RelTool(U36,0,0,-300), vExtMax, z1, tWeldGun\WObj:=wobjHtip;
		MoveL RelTool(U36,0,0,-30), vExtMax, z1, tWeldGun\WObj:=wobjHtip;
		PDispSet SRU36XYZ;
		ArcLStart U36, v100, smTU3031quick, wdTU3031quick\Weave:=wvTU3031quick, fine, tWeldGun\WObj:=wobjHtip;
		ArcL U37, v100, smTU3031quick, wdTU3031quick\Weave:=wvTU3031quick, z10, tWeldGun\WObj:=wobjHtip;
		ArcLEnd U38, v100, smTU3031quick, wdTU3031SLOW\Weave:=wvTU3031quick, z10, tWeldGun\WObj:=wobjHtip;
		PDispOff;
		MoveL RelTool(U36,0,0,-30), v200, z1, tWeldGun\WObj:=wobjHtip;
		MoveL RelTool(U36,0,0,-300), vExtMax, z1, tWeldGun\WObj:=wobjHtip;
		MoveJ AIRTOU30_2, vExtMax, z1, tWeldGun\WObj:=wobjHtip;
		MoveL RelTool(T36,0,0,-300), v200, z1, tWeldGun\WObj:=wobjHtip;
        SEARCHT36Y:
		MoveL Offs(SPTY36E,0,100,0), vExtMax, z1, tWeldGun\WObj:=wobjHtip;
		Search_1D SRT36Y, Offs(SPTY36E,0,20,0), SPTY36E, v100, tWeldGun\WObj:=wobjHtip\SchSpeed:=10;
		MoveL Offs(SPTY36E,0,150,0), vExtMax, z1, tWeldGun\WObj:=wobjHtip;
		SRT36XYZ.trans.x := SRT33X.trans.x;
		SRT36XYZ.trans.y := SRT36Y.trans.y;
		SRT36XYZ.trans.z := SRT33Z.trans.z;
        WaitTime\InPos, .1;
		MoveL RelTool(T36,0,0,-300), vExtMax, z1, tWeldGun\WObj:=wobjHtip;
		MoveL RelTool(T36,0,0,-30), v200, z1, tWeldGun\WObj:=wobjHtip;
		PDispSet SRT36XYZ;
		ArcLStart T36, v100, smTU3031quick, wdTU3031quick\Weave:=wvTU3031quick, fine, tWeldGun\WObj:=wobjHtip;
		ArcL T37, v100, smTU3031quick, wdTU3031quick\Weave:=wvTU3031quick, z10, tWeldGun\WObj:=wobjHtip;
		ArcLEnd T38, v100, smTU3031quick, wdTU3031SLOW\Weave:=wvTU3031quick, z10, tWeldGun\WObj:=wobjHtip;
		PDispOff;
		MoveL RelTool(T36,0,0,-30), v200, z1, tWeldGun\WObj:=wobjHtip;
		MoveL RelTool(T36,0,0,-300), vExtMax, z1, tWeldGun\WObj:=wobjHtip;
		MoveJ pjthomeSTA1zero, vCellSpeed, fine, tWeldGun\WObj:=wobj0;
		MoveJ AIRTOT30_1, vExtMax, z1, tWeldGun\WObj:=wobjHtip;
		MoveJ AIRTOT30_2, vExtMax, z1, tWeldGun\WObj:=wobjHtip;
		MoveJ RelTool(T30,50,0,-50), vExtMax, z1, tWeldGun\WObj:=wobjHtip;
		MoveL RelTool(T30,50,0,-50), v200, z1, tWeldGun\WObj:=wobjHtip;
		PDispSet SRT33XYZ;
		ArcLStart T32, v100, smTU3031, wdTU3031cover\Weave:=wvTU3031cover, fine, tWeldGun\WObj:=wobjHtip;
		ArcL T30, v100, smTU3031, wdTU3031cover\Weave:=wvTU3031cover, z1, tWeldGun\WObj:=wobjHtip;
		ArcLEnd T31, v100, smTU3031, wdTU3031cover\Weave:=wvTU3031cover, fine, tWeldGun\WObj:=wobjHtip;
		PDispOff;
		MoveL RelTool(T30,50,0,-50), v200, z1, tWeldGun\WObj:=wobjHtip;
        TPErase;
        TPWrite "NOW WORKING ON WELD 'U30'";
		MoveJ AIRTOT30_2, vExtMax, z1, tWeldGun\WObj:=wobjHtip;
		MoveJ AIRTOT30_1, vExtMax, z1, tWeldGun\WObj:=wobjHtip;
		MoveJ Offs(U32,300,-200,100), vExtMax, z5, tWeldGun\WObj:=wobjHtip;
		MoveL RelTool(U32,20,20,-30), v200, z1, tWeldGun\WObj:=wobjHtip;
		PDispSet SRU33XYZ;
		ArcLStart U32, v100, smTU3031, wdTU3031cover\Weave:=wvTU3031cover, fine, tWeldGun\WObj:=wobjHtip;
		ArcL U30, v100, smTU3031, wdTU3031cover\Weave:=wvTU3031cover, z1, tWeldGun\WObj:=wobjHtip;
		ArcLEnd U31, v100, smTU3031, wdTU3031cover\Weave:=wvTU3031cover, fine, tWeldGun\WObj:=wobjHtip;
		PDispOff;
		MoveL RelTool(U30,20,20,-30), v200, z1, tWeldGun\WObj:=wobjHtip;
		MoveJ Offs(U30,300,-200,100), vExtMax, z5, tWeldGun\WObj:=wobjHtip;
		SKIP_TU30s:
		MoveJ pjthomeSTA1zero, vCellSpeed, fine, tWeldGun\WObj:=wobj0;
		LABEL27:
	ENDPROC

	PROC WELDpivot_18H()
        !!!!NEW (18H) WELDpivot for PR3 04-08-18!!!!!
        !!!! has percentcoverpass!!!!!
        !CutWire;
	    ActUnit STN1;
	    AccSet 40, 40;
	    MoveJ pjthomeSTA1zero, vCellSpeed, fine, tWeldGun\WObj:=wobj0;
	    have_front_wrapper:
        IF pivCAM = FALSE THEN
           Piv_side_Welds "G";
           Piv_side_Welds "H";
        !!  THIS ONLY HAPPENS ON A NON CAM PIVOT CASTING
        ENDIF
        WELD_ALLPIV_PJ_18H "G" ;
        CutWire;
        WELD_ALLPIV_PJ_18H "H" ;
		MoveJ pjthomeSTA1zero, vCellSpeed, z5, tWeldGun\WObj:=wobj0;
		MoveJ Offs(T22,0,-200,150), vExtMax, z5, tWeldGun\WObj:=wobjHtip;
		MoveL SPT20S, v200, z5, tWeldGun\WObj:=wobjHtip;
        TPErase;
		Search_1D\Wire, SRT20, SPT20S, SPT20E, v100, tWeldGun\WObj:=wobjHtip\SchSpeed:=10;
        TPWrite "SRT20 XYZ:="\Pos:=SRT20.trans;
		MoveL SPT20S, v200, z5, tWeldGun\WObj:=wobjHtip;
		PDispSet SRT20;
        TPWrite "NOW WORKING ON WELD 'T20'";
		MoveL Offs(T22,0,-20,15), v100, z5, tWeldGun\WObj:=wobjHtip;
		ArcLStart T21, v100, smTU2122, wdTU2122cover\Weave:=wvTU2122cover, z1, tWeldGun\WObj:=wobjHtip;
		ArcL Offs(T21,3,0,0), v100, smTU2122, wdTU2122cover\Weave:=wvTU2122cover, z1, tWeldGun\WObj:=wobjHtip;
		ArcLEnd T22, v100, smTU2122, wdTU2122cover\Weave:=wvTU2122cover, z1, tWeldGun\WObj:=wobjHtip;
		MoveL Offs(T22,0,-20,15), v100, z5, tWeldGun\WObj:=wobjHtip;
		ArcLStart U21, v100, smTU2122, wdTU2122cover\Weave:=wvTU2122cover, z1, tWeldGun\WObj:=wobjHtip;
		ArcL Offs(U21,-3,0,0), v100, smTU2122, wdTU2122cover\Weave:=wvTU2122cover, z1, tWeldGun\WObj:=wobjHtip;
		ArcLEnd U22, v100, smTU2122, wdTU2122cover\Weave:=wvTU2122cover, z1, tWeldGun\WObj:=wobjHtip;
		PDispOff;
		MoveL Offs(U22,0,-20,15), vExtMax, z5, tWeldGun\WObj:=wobjHtip;
		MoveL Offs(U22,0,-180,55), vExtMax, z5, tWeldGun\WObj:=wobjHtip;
		MoveJ Offs(T22,0,-300,250), vExtMax, z5, tWeldGun\WObj:=wobjHtip;
		MoveJ pjthomeSTA1zero, vCellSpeed, fine, tWeldGun\WObj:=wobj0;
        GET_OUT:
   	ENDPROC

	PROC pausetoTACKBACKWRAP()
		MoveToPark;
		IF bUnderANCHOR = FALSE THEN
			GOTO stubborn2;
		ELSE
			GOTO don2;
		ENDIF
        stubborn2:
        ActUnit STN1;
        CellMoveJ pAtParkPos, v500, fine, tool0\WObj:=obCELL\ExtJointValues:=neg90;
        DeactUnit STN1;
		TPReadFK reg8, "REMEMBER to handweld any MISSING WELD around     the anchor?", stEmpty, "YES", "NO", stEmpty, stEmpty;
		IF reg8 = 2 THEN
			GOTO don2;
		ENDIF
		GOTO stubborn2;
		don2:
        ActUnit STN1;
        CellMoveJ pAtParkPos, v500, fine, tool0\WObj:=obCELL\ExtJointValues:=negzeroes;
		DeactUnit STN1;
        TPErase;
        TPWrite "                                          ";
        TPWrite "                                          ";
        TPWrite " TACK THE BACK WRAPPER TO THE SKELETON ";
        TPWrite " PRESS THE OP READY WHEN FINISHED ";
        TPWrite "                                          ";
        TPWrite "                                          ";
        TPWrite "                                          ";
        TPWrite "                                          ";
        waitfordi:
        WaitDI diSTN1_RDY_R1, 0;
        WaitTime 1;
        WaitDI diSTN1_RDY_R1, 1;
        !THE BACK WRAPPER BETTER BE ON
		TPErase;
		!!!!!!!THUS ENDS THE SKELETON>>> PUT ON THE WRAPPER
        TPErase;
        TPWrite "                                          ";
        TPWrite "                                          ";
        TPWrite "MOVING TO WELD THE REST OF ARM";
	    MoveToHome;
	    ActUnit STN1;
	    MoveJ pjthomeSTA1zero, vCellSpeed, fine, tWeldGun\WObj:=wobj0;
	    have_back_wrapper:
	ENDPROC

	PROC pausetoTACKFRONTWRAP()
		MoveToPark;
		TPErase;
		!!!!!!!THUS ENDS THE SKELETON>>> PUT ON THE WRAPPER
        ActUnit STN1;
        CellMoveJ pAtParkPos, v500, fine, tool0\WObj:=obCELL\ExtJointValues:=neg90;
        DeactUnit STN1;
        TPErase;
        TPWrite "                                          ";
        TPWrite " YOU MUST WELD THE FRONT of the ANCHOR";
        TPWrite " THE ROBOT MISSED TWO WELDS ON THE ANCHOR ";
		IF bmissweld = TRUE THEN
			GOTO stubborn2;
		ELSE
			GOTO don2;
		ENDIF
        stubborn2:
		TPReadFK reg8, "REMEMBER to handweld 2 missing WELDS in front     the anchor?", stEmpty, "YES", "NO", stEmpty, stEmpty;
		IF reg8 = 2 THEN
			GOTO don2;
		ENDIF
		GOTO stubborn2;
		don2:
        ActUnit STN1;
        CellMoveJ pAtParkPos, v500, fine, tool0\WObj:=obCELL\ExtJointValues:=neg180b;
		DeactUnit STN1;
        TPErase;
        TPWrite "                                          ";
        TPWrite " TACK THE FRONT WRAPPER TO THE SKELETON ";
        TPWrite " PRESS THE OP READY WHEN FINISHED ";
        waitfordihere:
        WaitDI diSTN1_RDY_R1, 0;
        WaitTime 1;
        WaitDI diSTN1_RDY_R1, 1;
        ActUnit STN1;
        CellMoveJ pAtParkPos, v500, fine, tool0\WObj:=obCELL\ExtJointValues:=negzeroes;
        !THE FRONT WRAPPER BETTER BE ON
        TPErase;
        TPWrite "                                          ";
        TPWrite "                                          ";
        TPWrite "MOVING TO WELD THE FRONT WRAPPER";
	    MoveToHome;
	ENDPROC

	PROC WELD_41_42_46s()
		ActUnit STN1;
    	AccSet 25, 25;
		MoveJ pjthomeSTA1zero, vCellSpeed, fine, tWeldGun\WObj:=wobj0;
        !!!! GETTING TO THE 3 Y SEARCHES FOR M 41,42,46!!!
		MoveJ YM41air1, vExtMax, z5, tWeldGun\WObj:=wobjHsideplate;
		MoveL YM41air2, vExtMax, z5, tWeldGun\WObj:=wobjHsideplate;
		MoveL p41air09, vExtMax, z5, tWeldGun\WObj:=wobjHsideplate;
		!MoveL RelTool(YM41S,180,0,-200), v500, z1, tWeldGun\WObj:=wobjHsideplate;
		MoveL RelTool(YM41S,0,0,0), v500, z1, tWeldGun\WObj:=wobjHsideplate;
		Search_1D SR_YZ_TEMP\SearchStop:=YZ_Temp, YM41S, YM41E, v300, tWeldGun\WObj:=wobjHsideplate\SchSpeed:=10;
        GHLM_YZ_POINT_SETTER M41, YZ_Temp, AA41;
        TPWrite "SRM41 XYZ:="\Pos:=SR_YZ_TEMP.trans;
        MoveL RelTool(YM41S,0,0,0), v500, z1, tWeldGun\WObj:=wobjHsideplate;
		Search_1D SR_YZ_TEMP\SearchStop:=YZ_Temp, YM42S, YM42E, v300, tWeldGun\WObj:=wobjHsideplate\SchSpeed:=10;
        GHLM_YZ_POINT_SETTER M42, YZ_Temp, AA42;
        TPWrite "SRM42 XYZ:="\Pos:=SR_YZ_TEMP.trans;
        MoveL RelTool(YM42S,0,0,0), v500, z1, tWeldGun\WObj:=wobjHsideplate;
		Search_1D SR_YZ_TEMP\SearchStop:=YZ_Temp, YM46S, YM46E, v300, tWeldGun\WObj:=wobjHsideplate\SchSpeed:=10;
        GHLM_YZ_POINT_SETTER M46, YZ_Temp, AA46;
        TPWrite "SRM46 XYZ:="\Pos:=SR_YZ_TEMP.trans;
        MoveL RelTool(YM46S,0,0,0), v500, z1, tWeldGun\WObj:=wobjHsideplate;
        !MoveL RelTool(YM41S,180,0,-100), v500, z1, tWeldGun\WObj:=wobjHsideplate;
		MoveL p41air09, vExtMax, z5, tWeldGun\WObj:=wobjHsideplate;
		MoveJ YM41air2, vExtMax, z5, tWeldGun\WObj:=wobjHsideplate;
		MoveJ YM41air1, vExtMax, z5, tWeldGun\WObj:=wobjHsideplate;
        SEARCH_Mx;
        SET_M40s_X;
        MoveJ Offs(M46,100,-250,0), vExtMax, z5, tWeldGun\WObj:=wobjHsideplate;
		MoveL RelTool(M42,0,0,-25), v100, z1, tWeldGun\WObj:=wobjHsideplate;
        TPErase;
        TPWrite "NOW WORKING ON WELD 'M40'";
		GOTO MPOINT3;
        !BELOW THIS LINE IS THE EDIT STRING FOR THE M41 L42 L46 BASEPOINTS
        PDispOff;
		MoveL RelTool(M41,0,0,-25), v100, z1, tWeldGun\WObj:=wobjHsideplate;
		MoveL M41, v100, z1, tWeldGun\WObj:=wobjHsideplate;
		MoveL RelTool(M42,0,0,-25), v100, z1, tWeldGun\WObj:=wobjHsideplate;
		MoveL M42, v100, z1, tWeldGun\WObj:=wobjHsideplate;
		MoveL RelTool(M46,0,0,-25), v100, z1, tWeldGun\WObj:=wobjHsideplate;
		MoveL M46, v100, z1, tWeldGun\WObj:=wobjHsideplate;
		MoveL RelTool(M46,0,0,-25), v100, z1, tWeldGun\WObj:=wobjHsideplate;
 		PDispOff;
 		SET_M40s_X;
		MoveL RelTool(M41,0,0,-25), v100, z1, tWeldGun\WObj:=wobjHsideplate;
        MPOINT3:
        MoveL RelTool(M41,0,0,-25), v100, z1, tWeldGun\WObj:=wobjHsideplate;
        MoveL RelTool(M41,0,0,-5), v100, z1, tWeldGun\WObj:=wobjHsideplate;
		ArcLStart M41, v100, smLM10, wdLM10\Weave:=wvLM10, fine, tWeldGun\WObj:=wobjHsideplate\Track:=trLM10;
		ArcCEnd M42, M46, v100, smLM10, wdLM10\Weave:=wvLM10, z5, tWeldGun\WObj:=wobjHsideplate\Track:=trLM10;
		MoveL RelTool(M46,0,0,-80), v100, z1, tWeldGun\WObj:=wobjHsideplate;
        TPErase;
		MoveJ Offs(M46,100,-250,0), vExtMax, z5, tWeldGun\WObj:=wobjHsideplate;
		MoveJ Offs(M46,300,-350,0), vExtMax, z5, tWeldGun\WObj:=wobjHsideplate;
        MoveJ Offs(L46,-100,-450,0), vExtMax, z5, tWeldGun\WObj:=wobjHsideplate;
        !!!! GETTING TO THE 3 Y SEARCHES FOR L 41,42,46!!!
        MoveJ YL41air1, vExtMax, z5, tWeldGun\WObj:=wobjHsideplate;
		MoveJ YL41air2, vExtMax, z5, tWeldGun\WObj:=wobjHsideplate;
		MoveJ RelTool(YL46S,-100,150,-100), v500, z1, tWeldGun\WObj:=wobjHsideplate;
		MoveJ RelTool(YL41S,-100,0,-100), v500, z1, tWeldGun\WObj:=wobjHsideplate;
		MoveL RelTool(YL41S,0,0,0), v500, z1, tWeldGun\WObj:=wobjHsideplate;
		Search_1D SR_YZ_TEMP\SearchStop:=YZ_Temp, YL41S, YL41E, v300, tWeldGun\WObj:=wobjHsideplate\SchSpeed:=10;
        GHLM_YZ_POINT_SETTER L41, YZ_Temp, AA41;
        TPWrite "SRL41 XYZ:="\Pos:=SR_YZ_TEMP.trans;
        MoveL RelTool(YL41S,0,0,0), v500, z1, tWeldGun\WObj:=wobjHsideplate;
			Search_1D SR_YZ_TEMP\SearchStop:=YZ_Temp, YL42S, YL42E, v300, tWeldGun\WObj:=wobjHsideplate\SchSpeed:=10;
        GHLM_YZ_POINT_SETTER L42, YZ_Temp, AA42;
        TPWrite "SRL42 XYZ:="\Pos:=SR_YZ_TEMP.trans;
        MoveL RelTool(YL42S,0,0,0), v500, z1, tWeldGun\WObj:=wobjHsideplate;
		Search_1D SR_YZ_TEMP\SearchStop:=YZ_Temp, YL46S, YL46E, v300, tWeldGun\WObj:=wobjHsideplate\SchSpeed:=10;
        GHLM_YZ_POINT_SETTER L46, YZ_Temp, AA46;
        TPWrite "SRL46 XYZ:="\Pos:=SR_YZ_TEMP.trans;
        MoveL RelTool(YL46S,-100,0,-100), v500, z1, tWeldGun\WObj:=wobjHsideplate;
        MoveJ RelTool(YL46S,-100,150,-100), vExtMax, z1, tWeldGun\WObj:=wobjHsideplate;
        MoveL RelTool(YL46S,-100,150,-300), v500, z1, tWeldGun\WObj:=wobjHsideplate;
        MoveL RelTool(YL46S,-100,550,-300), v500, z1, tWeldGun\WObj:=wobjHsideplate;
 		MoveL YL41air1, vExtMax, z5, tWeldGun\WObj:=wobjHsideplate;
        !!!!!!MOVING TO THE 3 X SEARCHES FOR L
		MoveJ halfwayhome_L, vExtMax, z1, tWeldGun\WObj:=wobjHsideplate;
        SEARCH_Lx;
        SET_L40s_X;
        MoveJ halfwayhome_L, vExtMax, z1, tWeldGun\WObj:=wobjHsideplate;
 		MoveL YL41air1, vExtMax, z5, tWeldGun\WObj:=wobjHsideplate;
 		PDispOff;
		MoveJ Offs(L46,-100,-450,0), vExtMax, z5, tWeldGun\WObj:=wobjHsideplate;
  		MoveL RelTool(L46,0,0,-80), v500, z1, tWeldGun\WObj:=wobjHsideplate;
		MoveL RelTool(L42,0,0,-25), v100, z1, tWeldGun\WObj:=wobjHsideplate;
        TPErase;
        TPWrite "NOW WORKING ON WELD 'L40'";
		GOTO LPOINT3;
        !BELOW THIS LINE IS THE EDIT STRING FOR THE L41 L42 L46 BASEPOINTS
        PDispOff;
		MoveL RelTool(L41,0,-50,-50), v100, z1, tWeldGun\WObj:=wobjHsideplate;
		MoveL L41, v100, z1, tWeldGun\WObj:=wobjHsideplate;
		MoveL RelTool(L42,0,0,-25), v100, z1, tWeldGun\WObj:=wobjHsideplate;
		MoveL L42, v100, z1, tWeldGun\WObj:=wobjHsideplate;
		MoveL RelTool(L46,0,0,-25), v100, z1, tWeldGun\WObj:=wobjHsideplate;
		MoveL L46, v100, z1, tWeldGun\WObj:=wobjHsideplate;
		MoveL RelTool(L46,0,0,-25), v100, z1, tWeldGun\WObj:=wobjHsideplate;
		PDispOff;
        SET_L40s_X;
		MoveL RelTool(L42,0,0,-50), v100, z1, tWeldGun\WObj:=wobjHsideplate;
        LPOINT3:
        MoveL RelTool(L42,0,0,-25), v100, z1, tWeldGun\WObj:=wobjHsideplate;
        MoveL RelTool(L41,0,0,-4), v100, fine, tWeldGun\WObj:=wobjHsideplate;
		ArcLStart L41, v100, smLM10, wdLM10\Weave:=wvLM10, fine, tWeldGun\WObj:=wobjHsideplate\Track:=trLM10;
		ArcCEnd L42, L46, v100, smLM10, wdLM10\Weave:=wvLM10, z5, tWeldGun\WObj:=wobjHsideplate\Track:=trLM10;
		MoveL RelTool(L46,0,0,-80), v100, z1, tWeldGun\WObj:=wobjHsideplate;
		MoveJ Offs(L46,-100,-250,0), vExtMax, z5, tWeldGun\WObj:=wobjHsideplate;
		MoveJ Offs(L46,-300,-350,0), vExtMax, z5, tWeldGun\WObj:=wobjHsideplate;
		MoveJ pjthomeSTA1zero, vCellSpeed, fine, tWeldGun\WObj:=wobj0;
        skippast:
	ENDPROC

	PROC WELD_49_47_45s()
		!THE BACK WRAPPER BETTER BE ON
		ActUnit STN1;
		AccSet 75, 75;
		MoveJ pjthomeSTA1zero, vCellSpeed, fine, tWeldGun\WObj:=wobj0;
        !!!! GETTING TO THE 4 Y SEARCHES FOR M 49,48,47,45!!!
		MoveJ YM41air1, vExtMax, z5, tWeldGun\WObj:=wobjHsideplate;
		MoveL YM41air2, vExtMax, z5, tWeldGun\WObj:=wobjHsideplate;
		MoveL RelTool(YM49S,0,400,0), v500, z1, tWeldGun\WObj:=wobjHsideplate;
		MoveL RelTool(YM49S,0,0,0), v500, z1, tWeldGun\WObj:=wobjHsideplate;
		Search_1D SR_YZ_TEMP\SearchStop:=YZ_Temp, YM49S, YM49E, v300, tWeldGun\WObj:=wobjHsideplate\SchSpeed:=10;
        GHLM_YZ_POINT_SETTER M49, YZ_Temp, AA49;
        TPWrite "SRM49 XYZ:="\Pos:=SR_YZ_TEMP.trans;
		MoveL RelTool(YM48S,0,0,0), v500, z1, tWeldGun\WObj:=wobjHsideplate;
		Search_1D SR_YZ_TEMP\SearchStop:=YZ_Temp, YM48S, YM48E, v300, tWeldGun\WObj:=wobjHsideplate\SchSpeed:=10;
        GHLM_YZ_POINT_SETTER M48, YZ_Temp, AA48;
        TPWrite "SRM48 XYZ:="\Pos:=SR_YZ_TEMP.trans;
        MoveL RelTool(YM48S,0,0,0), v500, z1, tWeldGun\WObj:=wobjHsideplate;
         Search_1D SR_YZ_TEMP\SearchStop:=YZ_Temp, YM47S, YM47E, v300, tWeldGun\WObj:=wobjHsideplate\SchSpeed:=10;
        GHLM_YZ_POINT_SETTER M47, YZ_Temp, AA47;
        TPWrite "SRM47 XYZ:="\Pos:=SR_YZ_TEMP.trans;
        MoveL RelTool(YM47S,0,0,0), v500, z1, tWeldGun\WObj:=wobjHsideplate;
		Search_1D SR_YZ_TEMP\SearchStop:=YZ_Temp, YM45S, YM45E, v300, tWeldGun\WObj:=wobjHsideplate\SchSpeed:=10;
        GHLM_YZ_POINT_SETTER M45, YZ_Temp, AA45;
        TPWrite "SRM45 XYZ:="\Pos:=SR_YZ_TEMP.trans;
        MoveL RelTool(YM45S,0,0,0), v500, z1, tWeldGun\WObj:=wobjHsideplate;
        MoveL RelTool(YM45S,150,0,0), v500, z1, tWeldGun\WObj:=wobjHsideplate;
		MoveJ YM41air2, vExtMax, z5, tWeldGun\WObj:=wobjHsideplate;
		MoveJ YM41air1, vExtMax, z5, tWeldGun\WObj:=wobjHsideplate;
		MoveJ RelTool(YM41air1,-150,0,-400), vExtMax, z5, tWeldGun\WObj:=wobjHsideplate;
		MoveJ halfwayhome_M, vCellSpeed, fine, tWeldGun\WObj:=wobjHsideplate;
        !!!! GETTING TO THE 1 X SEARCH FOR M 49,48,47,45!!!
        MoveJ Offs(XM49E,80,-400,0), vExtMax, fine, tWeldGun\WObj:=wobjHpivot;
        MoveL Offs(XM49E,80,0,0), vExtMax, fine, tWeldGun\WObj:=wobjHpivot;
		Search_1D SR_X_TEMP\SearchStop:=X_Temp, Offs(XM49E,30,0,0), XM49E, v300, tWeldGun\WObj:=wobjHpivot\SchSpeed:=10;
  		MoveL X_Temp, v50, fine, tWeldGun\WObj:=wobjHpivot;
        WaitTime\InPos, .2;
		Mx_weld_piv := CRobT(\Tool:=tWeldGun\WObj:=wobjHsideplate);
        TPWrite "SRM49X XYZ:="\Pos:=SR_X_TEMP.trans;
        MoveL Offs(XM49E,80,0,0), v500, z1, tWeldGun\WObj:=wobjHpivot;
		SET_M40s_X;
        MoveJ Offs(XM49E,80,-400,0), vExtMax, fine, tWeldGun\WObj:=wobjHpivot;
        !  THIS IS ADDED FOR PIVCAM
        IF pivCAM = TRUE THEN
           WELD_ALLPIV_1thru8 "G";
       ENDIF
        MoveJ RelTool(M49,0,-50,-250), vExtMax, z1, tWeldGun\WObj:=wobjHsideplate;
        MoveL RelTool(M49,0,0,-80), vExtMax, z1, tWeldGun\WObj:=wobjHsideplate;
        GOTO MPOINT2;
         !!!!!!!!!!!!!!THIS IS THE EDIT STRING FOR M 50,49,48,47,45!!!!!!!!!!
		MoveL RelTool(M49,0,0,-25), v100, z1, tWeldGun\WObj:=wobjHsideplate;
		MoveL M49, v100, z1, tWeldGun\WObj:=wobjHsideplate;
		MoveL M50, v100, z1, tWeldGun\WObj:=wobjHsideplate;
		MoveL M49, v100, z1, tWeldGun\WObj:=wobjHsideplate;
		MoveL M48, v100, z1, tWeldGun\WObj:=wobjHsideplate;
		MoveL RelTool(M47,0,0,-25), v100, z1, tWeldGun\WObj:=wobjHsideplate;
		MoveL M47, v100, z1, tWeldGun\WObj:=wobjHsideplate;
		MoveL RelTool(M45,0,0,-25), v100, z1, tWeldGun\WObj:=wobjHsideplate;
		MoveL M45, v100, z1, tWeldGun\WObj:=wobjHsideplate;
		MoveL RelTool(M45,0,0,-25), v100, z1, tWeldGun\WObj:=wobjHsideplate;
		SET_M40s_X;
		MoveL RelTool(M49,0,0,-80), v100, z1, tWeldGun\WObj:=wobjHsideplate;
        MPOINT2:
        TPErase;
        TPWrite "NOW WORKING ON WELD 'M'";
		ArcLStart RelTool(M50,2,0,-4), v100, smLM10, wdLM10\Weave:=wvLM10, fine, tWeldGun\WObj:=wobjHsideplate\Track:=trLM10;
		ArcL M49, v100, smLM10, wdLM10\Weave:=wvLM10, z5, tWeldGun\WObj:=wobjHsideplate\Track:=trLM10;
		ArcCEnd M47, M45, v100, smLM10, wdLM10\Weave:=wvLM10, z5, tWeldGun\WObj:=wobjHsideplate\Track:=trLM10;
		MoveL RelTool(M45,0,0,-80), v100, z1, tWeldGun\WObj:=wobjHsideplate;
		MoveJ Offs(M45,100,-250,150), vExtMax, z5, tWeldGun\WObj:=wobjHsideplate;
		MoveJ Offs(M45,300,-350,150), vExtMax, z5, tWeldGun\WObj:=wobjHsideplate;
		MoveJ Offs(L49,-300,-350,0), vExtMax, z5, tWeldGun\WObj:=wobjHsideplate;
        !!!! GETTING TO THE 4 Y SEARCHES FOR L 49,48,47,45!!!
        MoveL YL41air1, vExtMax, z5, tWeldGun\WObj:=wobjHsideplate;
		MoveJ YL41air2, vExtMax, z5, tWeldGun\WObj:=wobjHsideplate;
		MoveJ RelTool(YL49S,-150,-150,-80), vExtMax, z1, tWeldGun\WObj:=wobjHsideplate;
		MoveL RelTool(YL49S,0,0,0), v500, z1, tWeldGun\WObj:=wobjHsideplate;
		Search_1D SR_YZ_TEMP\SearchStop:=YZ_Temp, YL49S, YL49E, v300, tWeldGun\WObj:=wobjHsideplate\SchSpeed:=10;
        GHLM_YZ_POINT_SETTER L49, YZ_Temp, AA49;
        TPWrite "SRL49 XYZ:="\Pos:=SR_YZ_TEMP.trans;
        MoveL RelTool(YL48S,0,0,0), v500, z1, tWeldGun\WObj:=wobjHsideplate;
		Search_1D SR_YZ_TEMP\SearchStop:=YZ_Temp, YL48S, YL48E, v300, tWeldGun\WObj:=wobjHsideplate\SchSpeed:=10;
        GHLM_YZ_POINT_SETTER L48, YZ_Temp, AA48;
        TPWrite "SRL48 XYZ:="\Pos:=SR_YZ_TEMP.trans;
        MoveL RelTool(YL47S,0,0,0), v500, z1, tWeldGun\WObj:=wobjHsideplate;
         Search_1D SR_YZ_TEMP\SearchStop:=YZ_Temp, YL47S, YL47E, v300, tWeldGun\WObj:=wobjHsideplate\SchSpeed:=10;
        GHLM_YZ_POINT_SETTER L47, YZ_Temp, AA47;
        TPWrite "SRL47 XYZ:="\Pos:=SR_YZ_TEMP.trans;
        MoveJ RelTool(YL47S,0,0,0), v500, z1, tWeldGun\WObj:=wobjHsideplate;
         Search_1D SR_YZ_TEMP\SearchStop:=YZ_Temp, YL45S, YL45E, v300, tWeldGun\WObj:=wobjHsideplate\SchSpeed:=10;
        GHLM_YZ_POINT_SETTER L45, YZ_Temp, AA45;
        TPWrite "SRL45 XYZ:="\Pos:=SR_YZ_TEMP.trans;
        MoveL RelTool(YL45S,0,0,0), v500, z1, tWeldGun\WObj:=wobjHsideplate;
        MoveL RelTool(YL45S,-100,0,-100), v500, z1, tWeldGun\WObj:=wobjHsideplate;
        MoveL RelTool(YL45S,-100,0,-300), v500, z1, tWeldGun\WObj:=wobjHsideplate;
        !!!! GETTING TO THE 1 X SEARCH FOR L 49,48,47,45!!!
        MoveJ YL41air2, vExtMax, z5, tWeldGun\WObj:=wobjHsideplate;
        MoveJ XL4air23, vExtMax, z5, tWeldGun\WObj:=wobjHsideplate;
        MoveJ Offs(XL49E,120,0,50), v500, z1, tWeldGun\WObj:=wobjHpivot;
		MoveL Offs(XL49E,80,0,0), v500, z1, tWeldGun\WObj:=wobjHpivot;
        Search_1D SR_X_TEMP\SearchStop:=X_Temp, Offs(XL49E,30,0,0), XL49E, v300, tWeldGun\WObj:=wobjHpivot\SchSpeed:=10;
  		MoveL X_Temp, v50, fine, tWeldGun\WObj:=wobjHpivot;
        WaitTime\InPos, .2;
		Lx_weld_piv := CRobT(\Tool:=tWeldGun\WObj:=wobjHsideplate);
        TPWrite "SRL49X XYZ:="\Pos:=SR_X_TEMP.trans;
        MoveL Offs(XL49E,80,0,0), v500, z1, tWeldGun\WObj:=wobjHpivot;
        MoveL Offs(XL49E,120,0,50), v500, z1, tWeldGun\WObj:=wobjHpivot;
  		PDispOff;
        SET_L40s_X;
        MoveJ XL4air23, vExtMax, z5, tWeldGun\WObj:=wobjHsideplate;
        MoveJ YL41air2, vExtMax, z5, tWeldGun\WObj:=wobjHsideplate;
 		MoveL YL41air1, vExtMax, z5, tWeldGun\WObj:=wobjHsideplate;
        !MoveJ RelTool(L49,0,0,-250), vExtMax, z1, tWeldGun\WObj:=wobjHsideplate;
        IF pivCAM = TRUE THEN
           WELD_ALLPIV_1thru8 "H";
       ENDIF
        MoveL RelTool(L49,0,0,-80), vExtMax, z1, tWeldGun\WObj:=wobjHsideplate;
		GOTO LPOINT2;
         !!!!!!!!!!!!!!THIS IS THE EDIT STRING FOR L 50,49,48,47,45!!!!!!!!!!
		MoveL RelTool(L49,0,0,-25), v100, z1, tWeldGun\WObj:=wobjHsideplate;
		MoveL L49, v100, z1, tWeldGun\WObj:=wobjHsideplate;
		MoveL L50, v100, z1, tWeldGun\WObj:=wobjHsideplate;
		MoveL L49, v100, z1, tWeldGun\WObj:=wobjHsideplate;
		MoveL L48, v100, z1, tWeldGun\WObj:=wobjHsideplate;
		MoveL RelTool(L47,0,0,-25), v100, z1, tWeldGun\WObj:=wobjHsideplate;
		MoveL L47, v100, z1, tWeldGun\WObj:=wobjHsideplate;
		MoveL RelTool(L45,0,0,-25), v100, z1, tWeldGun\WObj:=wobjHsideplate;
		MoveL L45, v100, z1, tWeldGun\WObj:=wobjHsideplate;
		MoveL RelTool(L45,0,0,-25), v100, z1, tWeldGun\WObj:=wobjHsideplate;
		SET_L40s_X;
		MoveL RelTool(L49,0,0,-80), v100, z1, tWeldGun\WObj:=wobjHsideplate;
        LPOINT2:
        TPErase;
        TPWrite "NOW WORKING ON WELD 'L'";
		ArcLStart RelTool(L50,2,0,-5), v100, smLM10, wdLM10\Weave:=wvLM10, fine, tWeldGun\WObj:=wobjHsideplate\Track:=trLM10;
		ArcL L49, v100, smLM10, wdLM10\Weave:=wvLM10, z5, tWeldGun\WObj:=wobjHsideplate\Track:=trLM10;
		ArcCEnd L47, L45, v100, smLM10, wdLM10\Weave:=wvLM10, z5, tWeldGun\WObj:=wobjHsideplate\Track:=trLM10;
		MoveL RelTool(L45,0,0,-80), v100, z1, tWeldGun\WObj:=wobjHsideplate;
        TPErase;
		MoveL Offs(L45,-200,-250,150), vExtMax, z5, tWeldGun\WObj:=wobjHsideplate;
		MoveJ Offs(L45,-300,-350,150), vExtMax, z5, tWeldGun\WObj:=wobjHsideplate;
		MoveJ pjthomeSTA1zero, vCellSpeed, fine, tWeldGun\WObj:=wobj0;
		DONE:
	ENDPROC

	PROC FBadjpos()
        A395.extax.eax_b := FBfirst;
        A395L.extax.eax_b := FBfirst;
        A39.extax.eax_b := FBfirst;
        A38.extax.eax_b := FBfirst;
        A36.extax.eax_b := FBsecond;
        B395.extax.eax_b := FBfirst;
        B395L.extax.eax_b := FBfirst;
        B39.extax.eax_b := FBfirst;
        B38.extax.eax_b := FBfirst;
        B36.extax.eax_b := FBsecond;
        WaitTime\InPos, .2;
	ENDPROC

	PROC dripstop_G()
        G29.trans.y := G29.trans.y + scoot_G;
        G27.trans.y := G27.trans.y + scoot_G;
        G25.trans.y := G25.trans.y + scoot_G;
        G23.trans.y := G23.trans.y + scoot_G;
        G21.trans.y := G21.trans.y + scoot_G;
        G21K.trans.y := G21K.trans.y + scoot_G;
        G15K.trans.y := G15K.trans.y + scoot_G;
        G0.trans.y := G0.trans.y + scoot_G;
        G10.trans.y := G10.trans.y + scoot_G;
        G15.trans.y := G15.trans.y + scoot_G;
        G16.trans.y := G16.trans.y + scoot_G;
        G18.trans.y := G18.trans.y + scoot_G;
        G19.trans.y := G19.trans.y + scoot_G;
        WaitTime\InPos, .2;
	ENDPROC

	PROC dripstop_A()
        A39.trans.y := A39.trans.y + scoot_A;
        A38.trans.y := A38.trans.y + scoot_A;
        A37.trans.y := A37.trans.y + scoot_A;
        A35.trans.y := A35.trans.y + scoot_A;
        A36.trans.y := A36.trans.y + scoot_A;
        A36K.trans.y := A36K.trans.y + scoot_A;
        A33K.trans.y := A33K.trans.y + scoot_A;
        A34.trans.y := A34.trans.y + scoot_A;
        A33.trans.y := A33.trans.y + scoot_A;
        A32.trans.y := A32.trans.y + scoot_A;
        A325.trans.y := A325.trans.y + scoot_A;
        A31.trans.y := A31.trans.y + scoot_A;
        A30.trans.y := A30.trans.y + scoot_A;
        WaitTime\InPos, .2;
	ENDPROC

	PROC WELD_30s_ALL()
		ActUnit STN1;
		AccSet 75, 75;
		MoveJ pjthomeSTA1zero, vCellSpeed, fine, tWeldGun\WObj:=wobj0;
        TPErase;
        TPWrite "NOW WORKING ON THE FIRST HALF OF WELD 'A'";
		GOTO ASIDE1stSEGMENT;
        !!!!THIS IS THE ENTIRE "A" WELDS EDIT STRING IN CORRECT ORDER!!!!
        !!!!YOU CAN EDIT SEARCHES AND WELD POINTS HERE!!!!!!!!
        !!! GETTING IN POSITION FOR ALL Y SEARCHES ON THE A WELD
        !FBadjpos;
		MoveJ A39air1, vExtMax, z1, tWeldGun\WObj:=wobjHsideplate;
		MoveL RelTool(YA39S,-100,-100,-150), v500, z1, tWeldGun\WObj:=wobjHsideplate;
		Search_1D SR_YZ_TEMP\SearchStop:=YZ_Temp, YA39S, YA39E, v300, tWeldGun\WObj:=wobjHsideplate\SchSpeed:=10;
        AB_YZ_POINT_SETTER A39, YZ_Temp, AA39;
        TPWrite "SRA39 XYZ:="\Pos:=SR_YZ_TEMP.trans;
		MoveL RelTool(YA39S,0,0,0), v500, z1, tWeldGun\WObj:=wobjHsideplate;
		Search_1D SR_YZ_TEMP\SearchStop:=YZ_Temp, YA38S, YA38E, v300, tWeldGun\WObj:=wobjHsideplate\SchSpeed:=10;
        AB_YZ_POINT_SETTER A38, YZ_Temp, AA38;
        TPWrite "SRA38 XYZ:="\Pos:=SR_YZ_TEMP.trans;
		MoveL RelTool(YA38S,0,0,0), v500, z1, tWeldGun\WObj:=wobjHsideplate;
		Search_1D SR_YZ_TEMP\SearchStop:=YZ_Temp, YA36S, YA36E, v300, tWeldGun\WObj:=wobjHsideplate\SchSpeed:=10;
        AB_YZ_POINT_SETTER A36, YZ_Temp, AA36;
        TPWrite "SRA36 XYZ:="\Pos:=SR_YZ_TEMP.trans;
		MoveL RelTool(YA36S,0,0,0), v500, z1, tWeldGun\WObj:=wobjHsideplate;
		MoveL RelTool(YA36S,0,0,0), v500, z1, tWeldGun\WObj:=wobjHsideplate;
		Search_1D SR_YZ_TEMP\SearchStop:=YZ_Temp, YA33S, YA33E, v300, tWeldGun\WObj:=wobjHsideplate\SchSpeed:=10;
        AB_YZ_POINT_SETTER A33, YZ_Temp, AA33;
        TPWrite "SRA33 XYZ:="\Pos:=SR_YZ_TEMP.trans;
		MoveL RelTool(YA33S,0,0,0), v500, z1, tWeldGun\WObj:=wobjHsideplate;
		Search_1D SR_YZ_TEMP\SearchStop:=YZ_Temp, YA34S, YA34E, v300, tWeldGun\WObj:=wobjHsideplate\SchSpeed:=10;
        AB_YZ_POINT_SETTER A34, YZ_Temp, AA34;
        TPWrite "SRA34 XYZ:="\Pos:=SR_YZ_TEMP.trans;
		MoveL RelTool(YA34S,0,0,0), v500, z1, tWeldGun\WObj:=wobjHsideplate;
		Search_1D SR_YZ_TEMP\SearchStop:=YZ_Temp, YA32S, YA32E, v300, tWeldGun\WObj:=wobjHsideplate\SchSpeed:=10;
        AB_YZ_POINT_SETTER A32, YZ_Temp, AA32;
        TPWrite "SRA32 XYZ:="\Pos:=SR_YZ_TEMP.trans;
		MoveL RelTool(YA32S,0,0,0), v500, z1, tWeldGun\WObj:=wobjHsideplate;
		MoveL RelTool(YA30S,0,0,0), v500, z1, tWeldGun\WObj:=wobjHsideplate;
		Search_1D SR_YZ_TEMP\SearchStop:=YZ_Temp, YA30S, YA30E, v300, tWeldGun\WObj:=wobjHsideplate\SchSpeed:=10;
        AB_YZ_POINT_SETTER A30, YZ_Temp, AA30;
        TPWrite "SRA30 XYZ:="\Pos:=SR_YZ_TEMP.trans;
		MoveL RelTool(YA30S,0,0,0), v500, z1, tWeldGun\WObj:=wobjHsideplate;
		MoveL RelTool(YA33S,-100,0,-150), v500, z1, tWeldGun\WObj:=wobjHsideplate;
		MoveJ A39air1, vExtMax, z1, tWeldGun\WObj:=wobjHsideplate;
        SEARCH_Ax;
        SET_A30s_X;
		MoveJ RelTool(A39,0,0,-550), vExtMax, z1, tWeldGun\WObj:=wobjHsideplate;
		PDispOff;
		MoveL A395L, v100, z1, tWeldGun\WObj:=wobjHtip;
		MoveL A395, v100, z1, tWeldGun\WObj:=wobjHtip;
		MoveL A39, v100, z1, tWeldGun\WObj:=wobjHsideplate;
		MoveL A38, v100, z1, tWeldGun\WObj:=wobjHsideplate;
		MoveL A36, v100, z1, tWeldGun\WObj:=wobjHsideplate;
		MoveL A33, v100, z1, tWeldGun\WObj:=wobjHsideplate;
		MoveL RelTool(A34,0,0,-15), v100, z1, tWeldGun\WObj:=wobjHsideplate;
		MoveL A34, v100, z1, tWeldGun\WObj:=wobjHsideplate;
		MoveL RelTool(A32,0,0,-15), v100, z1, tWeldGun\WObj:=wobjHsideplate;
		MoveL A32, v100, z1, tWeldGun\WObj:=wobjHsideplate;
		MoveL RelTool(A30,0,0,-100), v100, z1, tWeldGun\WObj:=wobjHsideplate;
		MoveL RelTool(A30,0,0,-15), v100, z1, tWeldGun\WObj:=wobjHsideplate;
		MoveL A30, v100, z1, tWeldGun\WObj:=wobjHsideplate;
        SET_A30s_X;
		MoveL RelTool(A30,0,0,-25), v100, z1, tWeldGun\WObj:=wobjHsideplate;
		MoveL RelTool(A33,0,0,-50), v100, z1, tWeldGun\WObj:=wobjHsideplate;
		MoveL Offs(A395L,50,0,150), vExtMax, z5, tWeldGun\WObj:=wobjHtip;
        GOTO AROUND1st;
        ASIDE1stSEGMENT:
        !! GETTING IN POSITION FOR THE FIRST 3 Y SEARCHES ON THE A WELD
		MoveJ A39air1, vExtMax, z1, tWeldGun\WObj:=wobjHsideplate;
		MoveL RelTool(YA39S,-50,-70,-50), vExtMax, z1, tWeldGun\WObj:=wobjHsideplate;
		Search_1D SR_YZ_TEMP\SearchStop:=YZ_Temp, YA39S, YA39E, v300, tWeldGun\WObj:=wobjHsideplate\SchSpeed:=10;
        AB_YZ_POINT_SETTER A39, YZ_Temp, AA39;
        TPWrite "SRA39 XYZ:="\Pos:=SR_YZ_TEMP.trans;
		MoveL RelTool(YA39S,0,0,0), v500, z1, tWeldGun\WObj:=wobjHsideplate;
		Search_1D SR_YZ_TEMP\SearchStop:=YZ_Temp, YA38S, YA38E, v300, tWeldGun\WObj:=wobjHsideplate\SchSpeed:=10;
        AB_YZ_POINT_SETTER A38, YZ_Temp, AA38;
        TPWrite "SRA38 XYZ:="\Pos:=SR_YZ_TEMP.trans;
		MoveL RelTool(YA38S,0,0,0), v500, z1, tWeldGun\WObj:=wobjHsideplate;
		Search_1D SR_YZ_TEMP\SearchStop:=YZ_Temp, YA36S, YA36E, v300, tWeldGun\WObj:=wobjHsideplate\SchSpeed:=10;
        AB_YZ_POINT_SETTER A36, YZ_Temp, AA36;
        TPWrite "SRA36 XYZ:="\Pos:=SR_YZ_TEMP.trans;
		MoveL RelTool(YA36S,0,0,0), v500, z1, tWeldGun\WObj:=wobjHsideplate;
		MoveL RelTool(YA36S,0,0,0), v500, z1, tWeldGun\WObj:=wobjHsideplate;
		Search_1D SR_YZ_TEMP\SearchStop:=YZ_Temp, YA33S, YA33E, v300, tWeldGun\WObj:=wobjHsideplate\SchSpeed:=10;
        AB_YZ_POINT_SETTER A33, YZ_Temp, AA33;
        TPWrite "SRA33 XYZ:="\Pos:=SR_YZ_TEMP.trans;
		MoveL RelTool(YA33S,0,0,0), v500, z1, tWeldGun\WObj:=wobjHsideplate;		MoveJ A39air3, vExtMax, z1, tWeldGun\WObj:=wobjHsideplate;
		MoveJ A39air1, vExtMax, z1, tWeldGun\WObj:=wobjHsideplate;
        SEARCH_Ax;
        SET_A30s_X;
		MoveJ RelTool(A39,0,0,-350), vExtMax, z1, tWeldGun\WObj:=wobjHsideplate;
        AROUND1st:
        IF bWO458only = TRUE OR bWO459only = TRUE THEN
        dripstop_A;
        ENDIF
		MoveL Offs(A395L,20,0,20), vExtMax, z5, tWeldGun\WObj:=wobjHtip;
		ArcLStart A395L, v100, smGH195, wdGH195\Weave:=wvGH195, fine, tWeldGun\WObj:=wobjHtip\Track:=trABTBR;
		ArcL A395, v100, smGH195, wdGH195\Weave:=wvGH195, z1, tWeldGun\WObj:=wobjHtip\Track:=trABTBR;
		ArcL A38, v100, smGH195, wdGH195\Weave:=wvGH195, z1, tWeldGun\WObj:=wobjHsideplate\Track:=trABTBR;
		ArcCEnd A36, A33, v100, smGH195, wdGH195\Weave:=wvGH195, fine, tWeldGun\WObj:=wobjHsideplate\Track:=trABTBR;
		MoveL RelTool(A33,0,0,-50), vExtMax, z1, tWeldGun\WObj:=wobjHsideplate;
		MoveL RelTool(A33,0,0,-700), vExtMax, z1, tWeldGun\WObj:=wobjHsideplate;
		MoveJ pjthomeSTA1zero, vCellSpeed, fine, tWeldGun\WObj:=wobj0;
	    MoveJ RelTool(B33,0,0,-750), vExtMax, z1, tWeldGun\WObj:=wobjHsideplate;
        TPErase;
        TPWrite "NOW WORKING ON THE FIRST HALF OF WELD 'B'";
		GOTO BSIDE1stSEGMENT;
        !!!!THIS IS THE ENTIRE B SEARCHES EDIT STRING IN CORRECT ORDER!!!!
        !!!! GETTING IN POSITION FOR ALL Y SEARCHES ON THE B WELD
		MoveJ B39air2, vExtMax, z1, tWeldGun\WObj:=wobjHsideplate;
		MoveL RelTool(YB39S,0,100,-150), v500, z1, tWeldGun\WObj:=wobjHsideplate;
		Search_1D SR_YZ_TEMP\SearchStop:=YZ_Temp, YB39S, YB39E, v300, tWeldGun\WObj:=wobjHsideplate\SchSpeed:=10;
        AB_YZ_POINT_SETTER B39, YZ_Temp, AA39;
        TPWrite "SRB39 XYZ:="\Pos:=SR_YZ_TEMP.trans;
		MoveL RelTool(YB39S,0,0,0), v500, z1, tWeldGun\WObj:=wobjHsideplate;
		Search_1D SR_YZ_TEMP\SearchStop:=YZ_Temp, YB38S, YB38E, v300, tWeldGun\WObj:=wobjHsideplate\SchSpeed:=10;
        AB_YZ_POINT_SETTER B38, YZ_Temp, AA38;
        TPWrite "SRB38 XYZ:="\Pos:=SR_YZ_TEMP.trans;
		MoveL RelTool(YB38S,0,0,0), v500, z1, tWeldGun\WObj:=wobjHsideplate;
		Search_1D SR_YZ_TEMP\SearchStop:=YZ_Temp, YB36S, YB36E, v300, tWeldGun\WObj:=wobjHsideplate\SchSpeed:=10;
        AB_YZ_POINT_SETTER B36, YZ_Temp, AA36;
        TPWrite "SRB36 XYZ:="\Pos:=SR_YZ_TEMP.trans;
		MoveL RelTool(YB36S,0,0,0), v500, z1, tWeldGun\WObj:=wobjHsideplate;
		Search_1D SR_YZ_TEMP\SearchStop:=YZ_Temp, YB33S, YB33E, v300, tWeldGun\WObj:=wobjHsideplate\SchSpeed:=10;
        AB_YZ_POINT_SETTER B33, YZ_Temp, AA33;
        TPWrite "SRB33 XYZ:="\Pos:=SR_YZ_TEMP.trans;
		Search_1D SR_YZ_TEMP\SearchStop:=YZ_Temp, YB34S, YB34E, v300, tWeldGun\WObj:=wobjHsideplate\SchSpeed:=10;
        AB_YZ_POINT_SETTER B34, YZ_Temp, AA34;
        TPWrite "SRB34 XYZ:="\Pos:=SR_YZ_TEMP.trans;
		MoveL RelTool(YB34S,0,0,0), v500, z1, tWeldGun\WObj:=wobjHsideplate;
		MoveL RelTool(YB32S,0,50,0), v500, z1, tWeldGun\WObj:=wobjHsideplate;
		Search_1D SR_YZ_TEMP\SearchStop:=YZ_Temp, YB32S, YB32E, v300, tWeldGun\WObj:=wobjHsideplate\SchSpeed:=10;
        AB_YZ_POINT_SETTER B32, YZ_Temp, AA32;
        TPWrite "SRB32 XYZ:="\Pos:=SR_YZ_TEMP.trans;
		MoveL RelTool(YB32S,0,0,0), v500, z1, tWeldGun\WObj:=wobjHsideplate;
		MoveL RelTool(YB30S,0,50,0), v500, z1, tWeldGun\WObj:=wobjHsideplate;
		Search_1D SR_YZ_TEMP\SearchStop:=YZ_Temp, YB30S, YB30E, v300, tWeldGun\WObj:=wobjHsideplate\SchSpeed:=10;
        AB_YZ_POINT_SETTER B30, YZ_Temp, AA30;
        TPWrite "SRB30 XYZ:="\Pos:=SR_YZ_TEMP.trans;
		MoveL RelTool(YB30S,0,50,0), v500, z1, tWeldGun\WObj:=wobjHsideplate;
		MoveL RelTool(YB32S,0,50,0), v500, z1, tWeldGun\WObj:=wobjHsideplate;
		MoveL RelTool(YB33S,0,50,0), v500, z1, tWeldGun\WObj:=wobjHsideplate;
		MoveL RelTool(YB36S,0,50,0), v500, z1, tWeldGun\WObj:=wobjHsideplate;
		MoveJ B39air3, vExtMax, z1, tWeldGun\WObj:=wobjHsideplate;
		MoveJ B39air1, vExtMax, z1, tWeldGun\WObj:=wobjHsideplate;
        SEARCH_Bx;
        SET_B30s_X;
		MoveJ B39air1, vExtMax, z1, tWeldGun\WObj:=wobjHsideplate;
		MoveJ RelTool(B39,0,0,-350), vExtMax, z1, tWeldGun\WObj:=wobjHsideplate;
		MoveL B395L, v100, z1, tWeldGun\WObj:=wobjHtip;
		MoveL B395, v100, z1, tWeldGun\WObj:=wobjHtip;
		MoveL B39, v100, z1, tWeldGun\WObj:=wobjHsideplate;
		MoveL B38, v100, z1, tWeldGun\WObj:=wobjHsideplate;
		MoveL B36, v100, z1, tWeldGun\WObj:=wobjHsideplate;
		MoveL RelTool(B33,0,0,-15), v100, z1, tWeldGun\WObj:=wobjHsideplate;
		MoveL B33, v100, z1, tWeldGun\WObj:=wobjHsideplate;
		MoveL RelTool(B33,0,0,-15), v100, z1, tWeldGun\WObj:=wobjHsideplate;
		MoveL RelTool(B34,0,0,-15), v100, z1, tWeldGun\WObj:=wobjHsideplate;
		MoveL B34, v100, z1, tWeldGun\WObj:=wobjHsideplate;
		MoveL RelTool(B32,0,0,-15), v100, z1, tWeldGun\WObj:=wobjHsideplate;
		MoveL B32, v100, z1, tWeldGun\WObj:=wobjHsideplate;
		MoveL RelTool(B30,0,0,-135), v100, z1, tWeldGun\WObj:=wobjHsideplate;
		MoveL RelTool(B30,0,0,-15), v100, z1, tWeldGun\WObj:=wobjHsideplate;
		MoveL B30, v100, z1, tWeldGun\WObj:=wobjHsideplate;
        SET_B30s_X;
		MoveL RelTool(B32,0,0,-200), v100, z1, tWeldGun\WObj:=wobjHsideplate;
		MoveL RelTool(B33,0,0,-200), v100, z1, tWeldGun\WObj:=wobjHsideplate;
        GOTO BFIRSTTHIRD;
		BSIDE1stSEGMENT:
        !! GETTING IN POSITION FOR THE FIRST 3 Y SEARCHES ON THE B WELD
		MoveJ B39air2, vExtMax, z1, tWeldGun\WObj:=wobjHsideplate;
		MoveL RelTool(YB39S,0,100,-150), vExtMax, z1, tWeldGun\WObj:=wobjHsideplate;
		MoveL RelTool(YB39S,0,0,0), v500, z1, tWeldGun\WObj:=wobjHsideplate;
		Search_1D SR_YZ_TEMP\SearchStop:=YZ_Temp, YB39S, YB39E, v300, tWeldGun\WObj:=wobjHsideplate\SchSpeed:=10;
        AB_YZ_POINT_SETTER B39, YZ_Temp, AA39;
        TPWrite "SRB39 XYZ:="\Pos:=SR_YZ_TEMP.trans;
		MoveL RelTool(YB39S,0,0,0), v500, z1, tWeldGun\WObj:=wobjHsideplate;
		Search_1D SR_YZ_TEMP\SearchStop:=YZ_Temp, YB38S, YB38E, v300, tWeldGun\WObj:=wobjHsideplate\SchSpeed:=10;
        AB_YZ_POINT_SETTER B38, YZ_Temp, AA38;
        TPWrite "SRB38 XYZ:="\Pos:=SR_YZ_TEMP.trans;
		MoveL RelTool(YB38S,0,0,0), v500, z1, tWeldGun\WObj:=wobjHsideplate;
		Search_1D SR_YZ_TEMP\SearchStop:=YZ_Temp, YB36S, YB36E, v300, tWeldGun\WObj:=wobjHsideplate\SchSpeed:=10;
        AB_YZ_POINT_SETTER B36, YZ_Temp, AA36;
        TPWrite "SRB36 XYZ:="\Pos:=SR_YZ_TEMP.trans;
		MoveL RelTool(YB36S,0,0,0), v500, z1, tWeldGun\WObj:=wobjHsideplate;
		Search_1D SR_YZ_TEMP\SearchStop:=YZ_Temp, YB33S, YB33E, v300, tWeldGun\WObj:=wobjHsideplate\SchSpeed:=10;
        AB_YZ_POINT_SETTER B33, YZ_Temp, AA33;
        TPWrite "SRB33 XYZ:="\Pos:=SR_YZ_TEMP.trans;
		MoveL RelTool(YB33S,0,0,-150), v500, z1, tWeldGun\WObj:=wobjHsideplate;
		MoveJ B39air1, vExtMax, z1, tWeldGun\WObj:=wobjHsideplate;
        SEARCH_Bx;
        SET_B30s_X;
		MoveJ B39air1, vExtMax, z1, tWeldGun\WObj:=wobjHsideplate;
        BFIRSTTHIRD:
		MoveJ RelTool(B39,0,0,-350), vExtMax, z1, tWeldGun\WObj:=wobjHsideplate;
        SET_B30s_X;
		MoveJ RelTool(B395,0,0,-100), vExtMax, z1, tWeldGun\WObj:=wobjHtip;
		MoveL RelTool(B395,0,0,-50), vExtMax, z1, tWeldGun\WObj:=wobjHtip;
		ArcLStart B395L, v100, smGH195, wdGH195\Weave:=wvGH195, fine, tWeldGun\WObj:=wobjHtip\Track:=trAB;
		ArcL B395, v100, smGH195, wdGH195\Weave:=wvGH195, z1, tWeldGun\WObj:=wobjHtip\Track:=trAB;
		ArcL B38, v100, smGH195, wdGH195\Weave:=wvGH195, z1, tWeldGun\WObj:=wobjHsideplate\Track:=trAB;
		ArcCEnd B36, B33, v100, smGH195, wdGH195\Weave:=wvGH195, fine, tWeldGun\WObj:=wobjHsideplate\Track:=trAB;
		MoveL RelTool(B33,0,0,-50), vExtMax, z1, tWeldGun\WObj:=wobjHsideplate;
	    MoveL RelTool(B33,-200,0,-750), vExtMax, z1, tWeldGun\WObj:=wobjHsideplate;
	    MoveJ pjthomeSTA1zero, vCellSpeed, fine, tWeldGun\WObj:=wobj0;
        !!!GETTING IN POSITION FOR LAST 3 Y SEARCHES ON THE A WELD
        MoveJ RelTool(A33,0,0,-550), vExtMax, z1, tWeldGun\WObj:=wobjHsideplate;
		MoveL RelTool(YA33S,-150,0,-160), v500, z1, tWeldGun\WObj:=wobjHsideplate;
		MoveJ RelTool(YA30S,-100,0,0), vExtMax, z1, tWeldGun\WObj:=wobjHsideplate;
		Search_1D SR_YZ_TEMP\SearchStop:=YZ_Temp, YA30S, YA30E, v300, tWeldGun\WObj:=wobjHsideplate\SchSpeed:=10;
        AB_YZ_POINT_SETTER A30, YZ_Temp, AA30;
        TPWrite "SRA30 XYZ:="\Pos:=SR_YZ_TEMP.trans;
		MoveL RelTool(YA30S,0,0,0), v500, z1, tWeldGun\WObj:=wobjHsideplate;
		Search_1D SR_YZ_TEMP\SearchStop:=YZ_Temp, YA32S, YA32E, v300, tWeldGun\WObj:=wobjHsideplate\SchSpeed:=10;
        AB_YZ_POINT_SETTER A32, YZ_Temp, AA32;
        TPWrite "SRA32 XYZ:="\Pos:=SR_YZ_TEMP.trans;
		MoveL RelTool(YA32S,0,0,0), v500, z1, tWeldGun\WObj:=wobjHsideplate;
		Search_1D SR_YZ_TEMP\SearchStop:=YZ_Temp, YA34S, YA34E, v300, tWeldGun\WObj:=wobjHsideplate\SchSpeed:=10;
        AB_YZ_POINT_SETTER A34, YZ_Temp, AA34;
        TPWrite "SRA34 XYZ:="\Pos:=SR_YZ_TEMP.trans;
		MoveL RelTool(YA34S,0,0,0), v500, z1, tWeldGun\WObj:=wobjHsideplate;
		MoveL RelTool(YA34S,-150,0,-160), v500, z1, tWeldGun\WObj:=wobjHsideplate;
        !!!GETTING IN POSITION FOR LAST 3 X SEARCHES ON THE A WELD
		MoveJ A39air12, vExtMax, z1, tWeldGun\WObj:=wobjHsideplate;
        SEARCH_Ax;
        SET_A30s_X;
        TPErase;
        TPWrite "NOW WELDING ON LAST HALF OF WELD 'A'";
        IF bWO458only = TRUE OR bWO459only = TRUE THEN
        dripstop_A;
        ENDIF
		MoveJ RelTool(A30,0,0,-200), vExtMax, z1, tWeldGun\WObj:=wobjHsideplate;
		MoveL RelTool(A30,0,0,-50), vExtMax, z1, tWeldGun\WObj:=wobjHsideplate;
		ArcLStart RelTool(A30,0,-14,-1), v100, smGH195, wdGH195\Weave:=wvGH195, fine, tWeldGun\WObj:=wobjHsideplate\Track:=trABTBL;
		ArcCEnd A32, A34, v100, smGH195, wdGH195\Weave:=wvGH195, fine, tWeldGun\WObj:=wobjHsideplate\Track:=trABTBL;
		MoveL RelTool(A34,0,0,-150), vExtMax, z1, tWeldGun\WObj:=wobjHsideplate;
		MoveL RelTool(A34,0,0,-550), vExtMax, z1, tWeldGun\WObj:=wobjHsideplate;
		MoveJ RelTool(A34,0,0,-750), vExtMax, z1, tWeldGun\WObj:=wobjHsideplate;
		MoveJ pjthomeSTA1zero, vCellSpeed, fine, tWeldGun\WObj:=wobj0;
        !!!GETTING IN POSITION FOR LAST 3 Y SEARCHES ON THE B WELD
		MoveJ B30air1, vExtMax, z1, tWeldGun\WObj:=wobjHsideplate;
		MoveL RelTool(YB30S,0,70,-50), vExtMax, z1, tWeldGun\WObj:=wobjHsideplate;
		Search_1D SR_YZ_TEMP\SearchStop:=YZ_Temp, YB30S, YB30E, v300, tWeldGun\WObj:=wobjHsideplate\SchSpeed:=10;
        AB_YZ_POINT_SETTER B30, YZ_Temp, AA30;
        TPWrite "SRB30 XYZ:="\Pos:=SR_YZ_TEMP.trans;
		MoveL RelTool(YB30S,0,0,0), v500, z1, tWeldGun\WObj:=wobjHsideplate;
		Search_1D SR_YZ_TEMP\SearchStop:=YZ_Temp, YB32S, YB32E, v300, tWeldGun\WObj:=wobjHsideplate\SchSpeed:=10;
        AB_YZ_POINT_SETTER B32, YZ_Temp, AA32;
        TPWrite "SRB32 XYZ:="\Pos:=SR_YZ_TEMP.trans;
		MoveL RelTool(YB32S,0,0,0), v500, z1, tWeldGun\WObj:=wobjHsideplate;
		Search_1D SR_YZ_TEMP\SearchStop:=YZ_Temp, YB34S, YB34E, v300, tWeldGun\WObj:=wobjHsideplate\SchSpeed:=10;
        AB_YZ_POINT_SETTER B34, YZ_Temp, AA34;
        TPWrite "SRB34 XYZ:="\Pos:=SR_YZ_TEMP.trans;
		MoveL RelTool(YB34S,0,0,0), v500, z1, tWeldGun\WObj:=wobjHsideplate;
		MoveJ RelTool(YB34S,0,50,-150), v500, z1, tWeldGun\WObj:=wobjHsideplate;
		MoveL B30air1, vExtMax, z1, tWeldGun\WObj:=wobjHsideplate;
		MoveJ halfwayhome_B, v500, z1, tWeldGun\WObj:=wobjHsideplate;
        SEARCH_Bx;
        SET_B30s_X;
        TPWrite "NOW WORKING ON LAST HALF OF WELD 'B'";
        MoveJ halfwayhome_B, v500, z1, tWeldGun\WObj:=wobjHsideplate;
       	MoveL RelTool(B30,0,0,-150), vExtMax, z1, tWeldGun\WObj:=wobjHsideplate;
       	MoveL RelTool(B30,0,0,-50), vExtMax, z1, tWeldGun\WObj:=wobjHsideplate;
		ArcLStart RelTool(B30,0,-14,-1), v100, smGH195, wdGH195\Weave:=wvGH195, fine, tWeldGun\WObj:=wobjHsideplate\Track:=trAB;
		ArcCEnd B32, B34, v100, smGH195, wdGH195\Weave:=wvGH195, fine, tWeldGun\WObj:=wobjHsideplate\Track:=trAB;
		MoveL RelTool(B34,0,0,-100), vExtMax, z1, tWeldGun\WObj:=wobjHsideplate;
		MoveL RelTool(B34,-200,0,-550), vExtMax, z1, tWeldGun\WObj:=wobjHsideplate;
		MoveJ pjthomeSTA1zero, vCellSpeed, fine, tWeldGun\WObj:=wobj0;
        TPErase;
        TPWrite "DONE WELDING BACK WRAPPER THE track bias WAY";
    	THATSIT:
	ENDPROC

	PROC UNtilt19()
        UNTILT:
        G19.extax := G195.extax;
        H19.extax := H195.extax;
        WaitTime\InPos, .2;
	ENDPROC

